	UF : 1, UT : 1,		CONFIG : 'N U T, 0, 0, 1',
	X =  112.000  mm,	Y =  46.000  mm,	Z =   0.600 mm,
	W =180.000 deg,	P =   0.000 deg,	R =    90.000 deg
};
P[2787]{
   GP1:
	UF : 1, UT : 1,		CONFIG : 'N U T, 0, 0, 1',
	X =  112.000  mm,	Y =  46.000  mm,	Z =   15.000 mm,
	W =180.000 deg,	P =   0.000 deg,	R =    90.000 deg
};
P[2794]{
   GP1:
	UF : 1, UT : 1,		CONFIG : 'N U T, 0, 0, 1',
	X =  127.000  mm,	Y =  46.000  mm,	Z =   15.000 mm,
	W =180.000 deg,	P =   0.000 deg,	R =    90.000 deg
};
P[2795]{
   GP1:
	UF : 1, UT : 1,		CONFIG : 'N U T, 0, 0, 1',
	X =  127.000  mm,	Y =  46.000  mm,	Z =   0.600 mm,
	W =180.000 deg,	P =   0.000 deg,	R =    90.000 deg
};
P[2796]{
   GP1:
	UF : 1, UT : 1,		CONFIG : 'N U T, 0, 0, 1',
	X =  127.000  mm,	Y =  46.000  mm,	Z =   15.000 mm,
	W =180.000 deg,	P =   0.000 deg,	R =    90.000 deg
};
P[2797]{
   GP1:
	UF : 1, UT : 1,		CONFIG : 'N U T, 0, 0, 1',
	X =  130.000  mm,	Y =  46.000  mm,	Z =   15.000 mm,
	W =180.000 deg,	P =   0.000 deg,	R =    90.000 deg
};
P[2798]{
   GP1:
	UF : 1, UT : 1,		CONFIG : 'N U T, 0, 0, 1',
	X =  130.000  mm,	Y =  46.000  mm,	Z =   0.600 mm,
	W =180.000 deg,	P =   0.000 deg,	R =    90.000 deg
};
P[2799]{
   GP1:
	UF : 1, UT : 1,		CONFIG : 'N U T, 0, 0, 1',
	X =  130.000  mm,	Y =  46.000  mm,	Z =   15.000 mm,
	W =180.000 deg,	P =   0.000 deg,	R =    90.000 deg
};
P[2800]{
   GP1:
	UF : 1, UT : 1,		CONFIG : 'N U T, 0, 0, 1',
	X =  133.000  mm,	Y =  46.000  mm,	Z =   15.000 mm,
	W =180.000 deg,	P =   0.000 deg,	R =    90.000 deg
};
P[2801]{
   GP1:
	UF : 1, UT : 1,		CONFIG : 'N U T, 0, 0, 1',
	X =  133.000  mm,	Y =  46.000  mm,	Z =   0.600 mm,
	W =180.000 deg,	P =   0.000 deg,	R =    90.000 deg
};
P[2802]{
   GP1:
	UF : 1, UT : 1,		CONFIG : 'N U T, 0, 0, 1',
	X =  133.000  mm,	Y =  46.000  mm,	Z =   15.000 mm,
	W =180.000 deg,	P =   0.000 deg,	R =    90.000 deg
};
P[2806]{
   GP1:
	UF : 1, UT : 1,		CONFIG : 'N U T, 0, 0, 1',
	X =  139.000  mm,	Y =  46.000  mm,	Z =   15.000 mm,
	W =180.000 deg,	P =   0.000 deg,	R =    90.000 deg
};
P[2807]{
   GP1:
	UF : 1, UT : 1,		CONFIG : 'N U T, 0, 0, 1',
	X =  139.000  mm,	Y =  46.000  mm,	Z =   0.600 mm,
	W =180.000 deg,	P =   0.000 deg,	R =    90.000 deg
};
P[2808]{
   GP1:
	UF : 1, UT : 1,		CONFIG : 'N U T, 0, 0, 1',
	X =  139.000  mm,	Y =  46.000  mm,	Z =   15.000 mm,
	W =180.000 deg,	P =   0.000 deg,	R =    90.000 deg
};
P[2812]{
   GP1:
	UF : 1, UT : 1,		CONFIG : 'N U T, 0, 0, 1',
	X =  145.000  mm,	Y =  46.000  mm,	Z =   15.000 mm,
	W =180.000 deg,	P =   0.000 deg,	R =    90.000 deg
};
P[2813]{
   GP1:
	UF : 1, UT : 1,		CONFIG : 'N U T, 0, 0, 1',
	X =  145.000  mm,	Y =  46.000  mm,	Z =   0.600 mm,
	W =180.000 deg,	P =   0.000 deg,	R =    90.000 deg
};
P[2814]{
   GP1:
	UF : 1, UT : 1,		CONFIG : 'N U T, 0, 0, 1',
	X =  145.000  mm,	Y =  46.000  mm,	Z =   15.000 mm,
	W =180.000 deg,	P =   0.000 deg,	R =    90.000 deg
};
P[2824]{
   GP1:
	UF : 1, UT : 1,		CONFIG : 'N U T, 0, 0, 1',
	X =  175.000  mm,	Y =  46.000  mm,	Z =   15.000 mm,
	W =180.000 deg,	P =   0.000 deg,	R =    90.000 deg
};
P[2825]{
   GP1:
	UF : 1, UT : 1,		CONFIG : 'N U T, 0, 0, 1',
	X =  175.000  mm,	Y =  46.000  mm,	Z =   0.600 mm,
	W =180.000 deg,	P =   0.000 deg,	R =    90.000 deg
};
P[2826]{
   GP1:
	UF : 1, UT : 1,		CONFIG : 'N U T, 0, 0, 1',
	X =  175.000  mm,	Y =  46.000  mm,	Z =   15.000 mm,
	W =180.000 deg,	P =   0.000 deg,	R =    90.000 deg
};
P[2827]{
   GP1:
	UF : 1, UT : 1,		CONFIG : 'N U T, 0, 0, 1',
	X =  178.000  mm,	Y =  46.000  mm,	Z =   15.000 mm,
	W =180.000 deg,	P =   0.000 deg,	R =    90.000 deg
};
P[2828]{
   GP1:
	UF : 1, UT : 1,		CONFIG : 'N U T, 0, 0, 1',
	X =  178.000  mm,	Y =  46.000  mm,	Z =   0.600 mm,
	W =180.000 deg,	P =   0.000 deg,	R =    90.000 deg
};
P[2829]{
   GP1:
	UF : 1, UT : 1,		CONFIG : 'N U T, 0, 0, 1',
	X =  178.000  mm,	Y =  46.000  mm,	Z =   15.000 mm,
	W =180.000 deg,	P =   0.000 deg,	R =    90.000 deg
};
P[2830]{
   GP1:
	UF : 1, UT : 1,		CONFIG : 'N U T, 0, 0, 1',
	X =  1.000  mm,	Y =  49.000  mm,	Z =   15.000 mm,
	W =180.000 deg,	P =   0.000 deg,	R =    90.000 deg
};
P[2831]{
   GP1:
	UF : 1, UT : 1,		CONFIG : 'N U T, 0, 0, 1',
	X =  1.000  mm,	Y =  49.000  mm,	Z =   0.600 mm,
	W =180.000 deg,	P =   0.000 deg,	R =    90.000 deg
};
P[2832]{
   GP1:
	UF : 1, UT : 1,		CONFIG : 'N U T, 0, 0, 1',
	X =  1.000  mm,	Y =  49.000  mm,	Z =   15.000 mm,
	W =180.000 deg,	P =   0.000 deg,	R =    90.000 deg
};
P[2833]{
   GP1:
	UF : 1, UT : 1,		CONFIG : 'N U T, 0, 0, 1',
	X =  4.000  mm,	Y =  49.000  mm,	Z =   15.000 mm,
	W =180.000 deg,	P =   0.000 deg,	R =    90.000 deg
};
P[2834]{
   GP1:
	UF : 1, UT : 1,		CONFIG : 'N U T, 0, 0, 1',
	X =  4.000  mm,	Y =  49.000  mm,	Z =   0.600 mm,
	W =180.000 deg,	P =   0.000 deg,	R =    90.000 deg
};
P[2835]{
   GP1:
	UF : 1, UT : 1,		CONFIG : 'N U T, 0, 0, 1',
	X =  4.000  mm,	Y =  49.000  mm,	Z =   15.000 mm,
	W =180.000 deg,	P =   0.000 deg,	R =    90.000 deg
};
P[2836]{
   GP1:
	UF : 1, UT : 1,		CONFIG : 'N U T, 0, 0, 1',
	X =  7.000  mm,	Y =  49.000  mm,	Z =   15.000 mm,
	W =180.000 deg,	P =   0.000 deg,	R =    90.000 deg
};
P[2837]{
   GP1:
	UF : 1, UT : 1,		CONFIG : 'N U T, 0, 0, 1',
	X =  7.000  mm,	Y =  49.000  mm,	Z =   0.600 mm,
	W =180.000 deg,	P =   0.000 deg,	R =    90.000 deg
};
P[2838]{
   GP1:
	UF : 1, UT : 1,		CONFIG : 'N U T, 0, 0, 1',
	X =  7.000  mm,	Y =  49.000  mm,	Z =   15.000 mm,
	W =180.000 deg,	P =   0.000 deg,	R =    90.000 deg
};
P[2839]{
   GP1:
	UF : 1, UT : 1,		CONFIG : 'N U T, 0, 0, 1',
	X =  10.000  mm,	Y =  49.000  mm,	Z =   15.000 mm,
	W =180.000 deg,	P =   0.000 deg,	R =    90.000 deg
};
P[2840]{
   GP1:
	UF : 1, UT : 1,		CONFIG : 'N U T, 0, 0, 1',
	X =  10.000  mm,	Y =  49.000  mm,	Z =   0.600 mm,
	W =180.000 deg,	P =   0.000 deg,	R =    90.000 deg
};
P[2841]{
   GP1:
	UF : 1, UT : 1,		CONFIG : 'N U T, 0, 0, 1',
	X =  10.000  mm,	Y =  49.000  mm,	Z =   15.000 mm,
	W =180.000 deg,	P =   0.000 deg,	R =    90.000 deg
};
P[2842]{
   GP1:
	UF : 1, UT : 1,		CONFIG : 'N U T, 0, 0, 1',
	X =  13.000  mm,	Y =  49.000  mm,	Z =   15.000 mm,
	W =180.000 deg,	P =   0.000 deg,	R =    90.000 deg
};
P[2843]{
   GP1:
	UF : 1, UT : 1,		CONFIG : 'N U T, 0, 0, 1',
	X =  13.000  mm,	Y =  49.000  mm,	Z =   0.600 mm,
	W =180.000 deg,	P =   0.000 deg,	R =    90.000 deg
};
P[2844]{
   GP1:
	UF : 1, UT : 1,		CONFIG : 'N U T, 0, 0, 1',
	X =  13.000  mm,	Y =  49.000  mm,	Z =   15.000 mm,
	W =180.000 deg,	P =   0.000 deg,	R =    90.000 deg
};
P[2845]{
   GP1:
	UF : 1, UT : 1,		CONFIG : 'N U T, 0, 0, 1',
	X =  16.000  mm,	Y =  49.000  mm,	Z =   15.000 mm,
	W =180.000 deg,	P =   0.000 deg,	R =    90.000 deg
};
P[2846]{
   GP1:
	UF : 1, UT : 1,		CONFIG : 'N U T, 0, 0, 1',
	X =  16.000  mm,	Y =  49.000  mm,	Z =   0.600 mm,
	W =180.000 deg,	P =   0.000 deg,	R =    90.000 deg
};
P[2847]{
   GP1:
	UF : 1, UT : 1,		CONFIG : 'N U T, 0, 0, 1',
	X =  16.000  mm,	Y =  49.000  mm,	Z =   15.000 mm,
	W =180.000 deg,	P =   0.000 deg,	R =    90.000 deg
};
P[2848]{
   GP1:
	UF : 1, UT : 1,		CONFIG : 'N U T, 0, 0, 1',
	X =  19.000  mm,	Y =  49.000  mm,	Z =   15.000 mm,
	W =180.000 deg,	P =   0.000 deg,	R =    90.000 deg
};
P[2849]{
   GP1:
	UF : 1, UT : 1,		CONFIG : 'N U T, 0, 0, 1',
	X =  19.000  mm,	Y =  49.000  mm,	Z =   0.600 mm,
	W =180.000 deg,	P =   0.000 deg,	R =    90.000 deg
};
P[2850]{
   GP1:
	UF : 1, UT : 1,		CONFIG : 'N U T, 0, 0, 1',
	X =  19.000  mm,	Y =  49.000  mm,	Z =   15.000 mm,
	W =180.000 deg,	P =   0.000 deg,	R =    90.000 deg
};
P[2854]{
   GP1:
	UF : 1, UT : 1,		CONFIG : 'N U T, 0, 0, 1',
	X =  25.000  mm,	Y =  49.000  mm,	Z =   15.000 mm,
	W =180.000 deg,	P =   0.000 deg,	R =    90.000 deg
};
P[2855]{
   GP1:
	UF : 1, UT : 1,		CONFIG : 'N U T, 0, 0, 1',
	X =  25.000  mm,	Y =  49.000  mm,	Z =   0.600 mm,
	W =180.000 deg,	P =   0.000 deg,	R =    90.000 deg
};
P[2856]{
   GP1:
	UF : 1, UT : 1,		CONFIG : 'N U T, 0, 0, 1',
	X =  25.000  mm,	Y =  49.000  mm,	Z =   15.000 mm,
	W =180.000 deg,	P =   0.000 deg,	R =    90.000 deg
};
P[2857]{
   GP1:
	UF : 1, UT : 1,		CONFIG : 'N U T, 0, 0, 1',
	X =  28.000  mm,	Y =  49.000  mm,	Z =   15.000 mm,
	W =180.000 deg,	P =   0.000 deg,	R =    90.000 deg
};
P[2858]{
   GP1:
	UF : 1, UT : 1,		CONFIG : 'N U T, 0, 0, 1',
	X =  28.000  mm,	Y =  49.000  mm,	Z =   0.600 mm,
	W =180.000 deg,	P =   0.000 deg,	R =    90.000 deg
};
P[2859]{
   GP1:
	UF : 1, UT : 1,		CONFIG : 'N U T, 0, 0, 1',
	X =  28.000  mm,	Y =  49.000  mm,	Z =   15.000 mm,
	W =180.000 deg,	P =   0.000 deg,	R =    90.000 deg
};
P[2860]{
   GP1:
	UF : 1, UT : 1,		CONFIG : 'N U T, 0, 0, 1',
	X =  31.000  mm,	Y =  49.000  mm,	Z =   15.000 mm,
	W =180.000 deg,	P =   0.000 deg,	R =    90.000 deg
};
P[2861]{
   GP1:
	UF : 1, UT : 1,		CONFIG : 'N U T, 0, 0, 1',
	X =  31.000  mm,	Y =  49.000  mm,	Z =   0.600 mm,
	W =180.000 deg,	P =   0.000 deg,	R =    90.000 deg
};
P[2862]{
   GP1:
	UF : 1, UT : 1,		CONFIG : 'N U T, 0, 0, 1',
	X =  31.000  mm,	Y =  49.000  mm,	Z =   15.000 mm,
	W =180.000 deg,	P =   0.000 deg,	R =    90.000 deg
};
P[2863]{
   GP1:
	UF : 1, UT : 1,		CONFIG : 'N U T, 0, 0, 1',
	X =  34.000  mm,	Y =  49.000  mm,	Z =   15.000 mm,
	W =180.000 deg,	P =   0.000 deg,	R =    90.000 deg
};
P[2864]{
   GP1:
	UF : 1, UT : 1,		CONFIG : 'N U T, 0, 0, 1',
	X =  34.000  mm,	Y =  49.000  mm,	Z =   0.600 mm,
	W =180.000 deg,	P =   0.000 deg,	R =    90.000 deg
};
P[2865]{
   GP1:
	UF : 1, UT : 1,		CONFIG : 'N U T, 0, 0, 1',
	X =  34.000  mm,	Y =  49.000  mm,	Z =   15.000 mm,
	W =180.000 deg,	P =   0.000 deg,	R =    90.000 deg
};
P[2866]{
   GP1:
	UF : 1, UT : 1,		CONFIG : 'N U T, 0, 0, 1',
	X =  37.000  mm,	Y =  49.000  mm,	Z =   15.000 mm,
	W =180.000 deg,	P =   0.000 deg,	R =    90.000 deg
};
P[2867]{
   GP1:
	UF : 1, UT : 1,		CONFIG : 'N U T, 0, 0, 1',
	X =  37.000  mm,	Y =  49.000  mm,	Z =   0.600 mm,
	W =180.000 deg,	P =   0.000 deg,	R =    90.000 deg
};
P[2868]{
   GP1:
	UF : 1, UT : 1,		CONFIG : 'N U T, 0, 0, 1',
	X =  37.000  mm,	Y =  49.000  mm,	Z =   15.000 mm,
	W =180.000 deg,	P =   0.000 deg,	R =    90.000 deg
};
P[2869]{
   GP1:
	UF : 1, UT : 1,		CONFIG : 'N U T, 0, 0, 1',
	X =  40.000  mm,	Y =  49.000  mm,	Z =   15.000 mm,
	W =180.000 deg,	P =   0.000 deg,	R =    90.000 deg
};
P[2870]{
   GP1:
	UF : 1, UT : 1,		CONFIG : 'N U T, 0, 0, 1',
	X =  40.000  mm,	Y =  49.000  mm,	Z =   0.600 mm,
	W =180.000 deg,	P =   0.000 deg,	R =    90.000 deg
};
P[2871]{
   GP1:
	UF : 1, UT : 1,		CONFIG : 'N U T, 0, 0, 1',
	X =  40.000  mm,	Y =  49.000  mm,	Z =   15.000 mm,
	W =180.000 deg,	P =   0.000 deg,	R =    90.000 deg
};
P[2872]{
   GP1:
	UF : 1, UT : 1,		CONFIG : 'N U T, 0, 0, 1',
	X =  43.000  mm,	Y =  49.000  mm,	Z =   15.000 mm,
	W =180.000 deg,	P =   0.000 deg,	R =    90.000 deg
};
P[2873]{
   GP1:
	UF : 1, UT : 1,		CONFIG : 'N U T, 0, 0, 1',
	X =  43.000  mm,	Y =  49.000  mm,	Z =   0.600 mm,
	W =180.000 deg,	P =   0.000 deg,	R =    90.000 deg
};
P[2874]{
   GP1:
	UF : 1, UT : 1,		CONFIG : 'N U T, 0, 0, 1',
	X =  43.000  mm,	Y =  49.000  mm,	Z =   15.000 mm,
	W =180.000 deg,	P =   0.000 deg,	R =    90.000 deg
};
P[2875]{
   GP1:
	UF : 1, UT : 1,		CONFIG : 'N U T, 0, 0, 1',
	X =  46.000  mm,	Y =  49.000  mm,	Z =   15.000 mm,
	W =180.000 deg,	P =   0.000 deg,	R =    90.000 deg
};
P[2876]{
   GP1:
	UF : 1, UT : 1,		CONFIG : 'N U T, 0, 0, 1',
	X =  46.000  mm,	Y =  49.000  mm,	Z =   0.600 mm,
	W =180.000 deg,	P =   0.000 deg,	R =    90.000 deg
};
P[2877]{
   GP1:
	UF : 1, UT : 1,		CONFIG : 'N U T, 0, 0, 1',
	X =  46.000  mm,	Y =  49.000  mm,	Z =   15.000 mm,
	W =180.000 deg,	P =   0.000 deg,	R =    90.000 deg
};
P[2878]{
   GP1:
	UF : 1, UT : 1,		CONFIG : 'N U T, 0, 0, 1',
	X =  49.000  mm,	Y =  49.000  mm,	Z =   15.000 mm,
	W =180.000 deg,	P =   0.000 deg,	R =    90.000 deg
};
P[2879]{
   GP1:
	UF : 1, UT : 1,		CONFIG : 'N U T, 0, 0, 1',
	X =  49.000  mm,	Y =  49.000  mm,	Z =   0.600 mm,
	W =180.000 deg,	P =   0.000 deg,	R =    90.000 deg
};
P[2880]{
   GP1:
	UF : 1, UT : 1,		CONFIG : 'N U T, 0, 0, 1',
	X =  49.000  mm,	Y =  49.000  mm,	Z =   15.000 mm,
	W =180.000 deg,	P =   0.000 deg,	R =    90.000 deg
};
P[2881]{
   GP1:
	UF : 1, UT : 1,		CONFIG : 'N U T, 0, 0, 1',
	X =  52.000  mm,	Y =  49.000  mm,	Z =   15.000 mm,
	W =180.000 deg,	P =   0.000 deg,	R =    90.000 deg
};
P[2882]{
   GP1:
	UF : 1, UT : 1,		CONFIG : 'N U T, 0, 0, 1',
	X =  52.000  mm,	Y =  49.000  mm,	Z =   0.600 mm,
	W =180.000 deg,	P =   0.000 deg,	R =    90.000 deg
};
P[2883]{
   GP1:
	UF : 1, UT : 1,		CONFIG : 'N U T, 0, 0, 1',
	X =  52.000  mm,	Y =  49.000  mm,	Z =   15.000 mm,
	W =180.000 deg,	P =   0.000 deg,	R =    90.000 deg
};
P[2884]{
   GP1:
	UF : 1, UT : 1,		CONFIG : 'N U T, 0, 0, 1',
	X =  55.000  mm,	Y =  49.000  mm,	Z =   15.000 mm,
	W =180.000 deg,	P =   0.000 deg,	R =    90.000 deg
};
P[2885]{
   GP1:
	UF : 1, UT : 1,		CONFIG : 'N U T, 0, 0, 1',
	X =  55.000  mm,	Y =  49.000  mm,	Z =   0.600 mm,
	W =180.000 deg,	P =   0.000 deg,	R =    90.000 deg
};
P[2886]{
   GP1:
	UF : 1, UT : 1,		CONFIG : 'N U T, 0, 0, 1',
	X =  55.000  mm,	Y =  49.000  mm,	Z =   15.000 mm,
	W =180.000 deg,	P =   0.000 deg,	R =    90.000 deg
};
P[2887]{
   GP1:
	UF : 1, UT : 1,		CONFIG : 'N U T, 0, 0, 1',
	X =  58.000  mm,	Y =  49.000  mm,	Z =   15.000 mm,
	W =180.000 deg,	P =   0.000 deg,	R =    90.000 deg
};
P[2888]{
   GP1:
	UF : 1, UT : 1,		CONFIG : 'N U T, 0, 0, 1',
	X =  58.000  mm,	Y =  49.000  mm,	Z =   0.600 mm,
	W =180.000 deg,	P =   0.000 deg,	R =    90.000 deg
};
P[2889]{
   GP1:
	UF : 1, UT : 1,		CONFIG : 'N U T, 0, 0, 1',
	X =  58.000  mm,	Y =  49.000  mm,	Z =   15.000 mm,
	W =180.000 deg,	P =   0.000 deg,	R =    90.000 deg
};
P[2899]{
   GP1:
	UF : 1, UT : 1,		CONFIG : 'N U T, 0, 0, 1',
	X =  70.000  mm,	Y =  49.000  mm,	Z =   15.000 mm,
	W =180.000 deg,	P =   0.000 deg,	R =    90.000 deg
};
P[2900]{
   GP1:
	UF : 1, UT : 1,		CONFIG : 'N U T, 0, 0, 1',
	X =  70.000  mm,	Y =  49.000  mm,	Z =   0.600 mm,
	W =180.000 deg,	P =   0.000 deg,	R =    90.000 deg
};
P[2901]{
   GP1:
	UF : 1, UT : 1,		CONFIG : 'N U T, 0, 0, 1',
	X =  70.000  mm,	Y =  49.000  mm,	Z =   15.000 mm,
	W =180.000 deg,	P =   0.000 deg,	R =    90.000 deg
};
P[2902]{
   GP1:
	UF : 1, UT : 1,		CONFIG : 'N U T, 0, 0, 1',
	X =  73.000  mm,	Y =  49.000  mm,	Z =   15.000 mm,
	W =180.000 deg,	P =   0.000 deg,	R =    90.000 deg
};
P[2903]{
   GP1:
	UF : 1, UT : 1,		CONFIG : 'N U T, 0, 0, 1',
	X =  73.000  mm,	Y =  49.000  mm,	Z =   0.600 mm,
	W =180.000 deg,	P =   0.000 deg,	R =    90.000 deg
};
P[2904]{
   GP1:
	UF : 1, UT : 1,		CONFIG : 'N U T, 0, 0, 1',
	X =  73.000  mm,	Y =  49.000  mm,	Z =   15.000 mm,
	W =180.000 deg,	P =   0.000 deg,	R =    90.000 deg
};
P[2905]{
   GP1:
	UF : 1, UT : 1,		CONFIG : 'N U T, 0, 0, 1',
	X =  76.000  mm,	Y =  49.000  mm,	Z =   15.000 mm,
	W =180.000 deg,	P =   0.000 deg,	R =    90.000 deg
};
P[2906]{
   GP1:
	UF : 1, UT : 1,		CONFIG : 'N U T, 0, 0, 1',
	X =  76.000  mm,	Y =  49.000  mm,	Z =   0.600 mm,
	W =180.000 deg,	P =   0.000 deg,	R =    90.000 deg
};
P[2907]{
   GP1:
	UF : 1, UT : 1,		CONFIG : 'N U T, 0, 0, 1',
	X =  76.000  mm,	Y =  49.000  mm,	Z =   15.000 mm,
	W =180.000 deg,	P =   0.000 deg,	R =    90.000 deg
};
P[2917]{
   GP1:
	UF : 1, UT : 1,		CONFIG : 'N U T, 0, 0, 1',
	X =  88.000  mm,	Y =  49.000  mm,	Z =   15.000 mm,
	W =180.000 deg,	P =   0.000 deg,	R =    90.000 deg
};
P[2918]{
   GP1:
	UF : 1, UT : 1,		CONFIG : 'N U T, 0, 0, 1',
	X =  88.000  mm,	Y =  49.000  mm,	Z =   0.600 mm,
	W =180.000 deg,	P =   0.000 deg,	R =    90.000 deg
};
P[2919]{
   GP1:
	UF : 1, UT : 1,		CONFIG : 'N U T, 0, 0, 1',
	X =  88.000  mm,	Y =  49.000  mm,	Z =   15.000 mm,
	W =180.000 deg,	P =   0.000 deg,	R =    90.000 deg
};
P[2920]{
   GP1:
	UF : 1, UT : 1,		CONFIG : 'N U T, 0, 0, 1',
	X =  91.000  mm,	Y =  49.000  mm,	Z =   15.000 mm,
	W =180.000 deg,	P =   0.000 deg,	R =    90.000 deg
};
P[2921]{
   GP1:
	UF : 1, UT : 1,		CONFIG : 'N U T, 0, 0, 1',
	X =  91.000  mm,	Y =  49.000  mm,	Z =   0.600 mm,
	W =180.000 deg,	P =   0.000 deg,	R =    90.000 deg
};
P[2922]{
   GP1:
	UF : 1, UT : 1,		CONFIG : 'N U T, 0, 0, 1',
	X =  91.000  mm,	Y =  49.000  mm,	Z =   15.000 mm,
	W =180.000 deg,	P =   0.000 deg,	R =    90.000 deg
};
P[2923]{
   GP1:
	UF : 1, UT : 1,		CONFIG : 'N U T, 0, 0, 1',
	X =  94.000  mm,	Y =  49.000  mm,	Z =   15.000 mm,
	W =180.000 deg,	P =   0.000 deg,	R =    90.000 deg
};
P[2924]{
   GP1:
	UF : 1, UT : 1,		CONFIG : 'N U T, 0, 0, 1',
	X =  94.000  mm,	Y =  49.000  mm,	Z =   0.600 mm,
	W =180.000 deg,	P =   0.000 deg,	R =    90.000 deg
};
P[2925]{
   GP1:
	UF : 1, UT : 1,		CONFIG : 'N U T, 0, 0, 1',
	X =  94.000  mm,	Y =  49.000  mm,	Z =   15.000 mm,
	W =180.000 deg,	P =   0.000 deg,	R =    90.000 deg
};
P[2926]{
   GP1:
	UF : 1, UT : 1,		CONFIG : 'N U T, 0, 0, 1',
	X =  97.000  mm,	Y =  49.000  mm,	Z =   15.000 mm,
	W =180.000 deg,	P =   0.000 deg,	R =    90.000 deg
};
P[2927]{
   GP1:
	UF : 1, UT : 1,		CONFIG : 'N U T, 0, 0, 1',
	X =  97.000  mm,	Y =  49.000  mm,	Z =   0.600 mm,
	W =180.000 deg,	P =   0.000 deg,	R =    90.000 deg
};
P[2928]{
   GP1:
	UF : 1, UT : 1,		CONFIG : 'N U T, 0, 0, 1',
	X =  97.000  mm,	Y =  49.000  mm,	Z =   15.000 mm,
	W =180.000 deg,	P =   0.000 deg,	R =    90.000 deg
};
P[2929]{
   GP1:
	UF : 1, UT : 1,		CONFIG : 'N U T, 0, 0, 1',
	X =  100.000  mm,	Y =  49.000  mm,	Z =   15.000 mm,
	W =180.000 deg,	P =   0.000 deg,	R =    90.000 deg
};
P[2930]{
   GP1:
	UF : 1, UT : 1,		CONFIG : 'N U T, 0, 0, 1',
	X =  100.000  mm,	Y =  49.000  mm,	Z =   0.600 mm,
	W =180.000 deg,	P =   0.000 deg,	R =    90.000 deg
};
P[2931]{
   GP1:
	UF : 1, UT : 1,		CONFIG : 'N U T, 0, 0, 1',
	X =  100.000  mm,	Y =  49.000  mm,	Z =   15.000 mm,
	W =180.000 deg,	P =   0.000 deg,	R =    90.000 deg
};
P[2932]{
   GP1:
	UF : 1, UT : 1,		CONFIG : 'N U T, 0, 0, 1',
	X =  103.000  mm,	Y =  49.000  mm,	Z =   15.000 mm,
	W =180.000 deg,	P =   0.000 deg,	R =    90.000 deg
};
P[2933]{
   GP1:
	UF : 1, UT : 1,		CONFIG : 'N U T, 0, 0, 1',
	X =  103.000  mm,	Y =  49.000  mm,	Z =   0.600 mm,
	W =180.000 deg,	P =   0.000 deg,	R =    90.000 deg
};
P[2934]{
   GP1:
	UF : 1, UT : 1,		CONFIG : 'N U T, 0, 0, 1',
	X =  103.000  mm,	Y =  49.000  mm,	Z =   15.000 mm,
	W =180.000 deg,	P =   0.000 deg,	R =    90.000 deg
};
P[2935]{
   GP1:
	UF : 1, UT : 1,		CONFIG : 'N U T, 0, 0, 1',
	X =  106.000  mm,	Y =  49.000  mm,	Z =   15.000 mm,
	W =180.000 deg,	P =   0.000 deg,	R =    90.000 deg
};
P[2936]{
   GP1:
	UF : 1, UT : 1,		CONFIG : 'N U T, 0, 0, 1',
	X =  106.000  mm,	Y =  49.000  mm,	Z =   0.600 mm,
	W =180.000 deg,	P =   0.000 deg,	R =    90.000 deg
};
P[2937]{
   GP1:
	UF : 1, UT : 1,		CONFIG : 'N U T, 0, 0, 1',
	X =  106.000  mm,	Y =  49.000  mm,	Z =   15.000 mm,
	W =180.000 deg,	P =   0.000 deg,	R =    90.000 deg
};
P[2938]{
   GP1:
	UF : 1, UT : 1,		CONFIG : 'N U T, 0, 0, 1',
	X =  109.000  mm,	Y =  49.000  mm,	Z =   15.000 mm,
	W =180.000 deg,	P =   0.000 deg,	R =    90.000 deg
};
P[2939]{
   GP1:
	UF : 1, UT : 1,		CONFIG : 'N U T, 0, 0, 1',
	X =  109.000  mm,	Y =  49.000  mm,	Z =   0.600 mm,
	W =180.000 deg,	P =   0.000 deg,	R =    90.000 deg
};
P[2940]{
   GP1:
	UF : 1, UT : 1,		CONFIG : 'N U T, 0, 0, 1',
	X =  109.000  mm,	Y =  49.000  mm,	Z =   15.000 mm,
	W =180.000 deg,	P =   0.000 deg,	R =    90.000 deg
};
P[2941]{
   GP1:
	UF : 1, UT : 1,		CONFIG : 'N U T, 0, 0, 1',
	X =  112.000  mm,	Y =  49.000  mm,	Z =   15.000 mm,
	W =180.000 deg,	P =   0.000 deg,	R =    90.000 deg
};
P[2942]{
   GP1:
	UF : 1, UT : 1,		CONFIG : 'N U T, 0, 0, 1',
	X =  112.000  mm,	Y =  49.000  mm,	Z =   0.600 mm,
	W =180.000 deg,	P =   0.000 deg,	R =    90.000 deg
};
P[2943]{
   GP1:
	UF : 1, UT : 1,		CONFIG : 'N U T, 0, 0, 1',
	X =  112.000  mm,	Y =  49.000  mm,	Z =   15.000 mm,
	W =180.000 deg,	P =   0.000 deg,	R =    90.000 deg
};
P[2950]{
   GP1:
	UF : 1, UT : 1,		CONFIG : 'N U T, 0, 0, 1',
	X =  127.000  mm,	Y =  49.000  mm,	Z =   15.000 mm,
	W =180.000 deg,	P =   0.000 deg,	R =    90.000 deg
};
P[2951]{
   GP1:
	UF : 1, UT : 1,		CONFIG : 'N U T, 0, 0, 1',
	X =  127.000  mm,	Y =  49.000  mm,	Z =   0.600 mm,
	W =180.000 deg,	P =   0.000 deg,	R =    90.000 deg
};
P[2952]{
   GP1:
	UF : 1, UT : 1,		CONFIG : 'N U T, 0, 0, 1',
	X =  127.000  mm,	Y =  49.000  mm,	Z =   15.000 mm,
	W =180.000 deg,	P =   0.000 deg,	R =    90.000 deg
};
P[2953]{
   GP1:
	UF : 1, UT : 1,		CONFIG : 'N U T, 0, 0, 1',
	X =  130.000  mm,	Y =  49.000  mm,	Z =   15.000 mm,
	W =180.000 deg,	P =   0.000 deg,	R =    90.000 deg
};
P[2954]{
   GP1:
	UF : 1, UT : 1,		CONFIG : 'N U T, 0, 0, 1',
	X =  130.000  mm,	Y =  49.000  mm,	Z =   0.600 mm,
	W =180.000 deg,	P =   0.000 deg,	R =    90.000 deg
};
P[2955]{
   GP1:
	UF : 1, UT : 1,		CONFIG : 'N U T, 0, 0, 1',
	X =  130.000  mm,	Y =  49.000  mm,	Z =   15.000 mm,
	W =180.000 deg,	P =   0.000 deg,	R =    90.000 deg
};
P[2959]{
   GP1:
	UF : 1, UT : 1,		CONFIG : 'N U T, 0, 0, 1',
	X =  136.000  mm,	Y =  49.000  mm,	Z =   15.000 mm,
	W =180.000 deg,	P =   0.000 deg,	R =    90.000 deg
};
P[2960]{
   GP1:
	UF : 1, UT : 1,		CONFIG : 'N U T, 0, 0, 1',
	X =  136.000  mm,	Y =  49.000  mm,	Z =   0.600 mm,
	W =180.000 deg,	P =   0.000 deg,	R =    90.000 deg
};
P[2961]{
   GP1:
	UF : 1, UT : 1,		CONFIG : 'N U T, 0, 0, 1',
	X =  136.000  mm,	Y =  49.000  mm,	Z =   15.000 mm,
	W =180.000 deg,	P =   0.000 deg,	R =    90.000 deg
};
P[2965]{
   GP1:
	UF : 1, UT : 1,		CONFIG : 'N U T, 0, 0, 1',
	X =  142.000  mm,	Y =  49.000  mm,	Z =   15.000 mm,
	W =180.000 deg,	P =   0.000 deg,	R =    90.000 deg
};
P[2966]{
   GP1:
	UF : 1, UT : 1,		CONFIG : 'N U T, 0, 0, 1',
	X =  142.000  mm,	Y =  49.000  mm,	Z =   0.600 mm,
	W =180.000 deg,	P =   0.000 deg,	R =    90.000 deg
};
P[2967]{
   GP1:
	UF : 1, UT : 1,		CONFIG : 'N U T, 0, 0, 1',
	X =  142.000  mm,	Y =  49.000  mm,	Z =   15.000 mm,
	W =180.000 deg,	P =   0.000 deg,	R =    90.000 deg
};
P[2986]{
   GP1:
	UF : 1, UT : 1,		CONFIG : 'N U T, 0, 0, 1',
	X =  175.000  mm,	Y =  49.000  mm,	Z =   15.000 mm,
	W =180.000 deg,	P =   0.000 deg,	R =    90.000 deg
};
P[2987]{
   GP1:
	UF : 1, UT : 1,		CONFIG : 'N U T, 0, 0, 1',
	X =  175.000  mm,	Y =  49.000  mm,	Z =   0.600 mm,
	W =180.000 deg,	P =   0.000 deg,	R =    90.000 deg
};
P[2988]{
   GP1:
	UF : 1, UT : 1,		CONFIG : 'N U T, 0, 0, 1',
	X =  175.000  mm,	Y =  49.000  mm,	Z =   15.000 mm,
	W =180.000 deg,	P =   0.000 deg,	R =    90.000 deg
};
P[2989]{
   GP1:
	UF : 1, UT : 1,		CONFIG : 'N U T, 0, 0, 1',
	X =  178.000  mm,	Y =  49.000  mm,	Z =   15.000 mm,
	W =180.000 deg,	P =   0.000 deg,	R =    90.000 deg
};
P[2990]{
   GP1:
	UF : 1, UT : 1,		CONFIG : 'N U T, 0, 0, 1',
	X =  178.000  mm,	Y =  49.000  mm,	Z =   0.600 mm,
	W =180.000 deg,	P =   0.000 deg,	R =    90.000 deg
};
P[2991]{
   GP1:
	UF : 1, UT : 1,		CONFIG : 'N U T, 0, 0, 1',
	X =  178.000  mm,	Y =  49.000  mm,	Z =   15.000 mm,
	W =180.000 deg,	P =   0.000 deg,	R =    90.000 deg
};
P[2992]{
   GP1:
	UF : 1, UT : 1,		CONFIG : 'N U T, 0, 0, 1',
	X =  1.000  mm,	Y =  52.000  mm,	Z =   15.000 mm,
	W =180.000 deg,	P =   0.000 deg,	R =    90.000 deg
};
P[2993]{
   GP1:
	UF : 1, UT : 1,		CONFIG : 'N U T, 0, 0, 1',
	X =  1.000  mm,	Y =  52.000  mm,	Z =   0.600 mm,
	W =180.000 deg,	P =   0.000 deg,	R =    90.000 deg
};
P[2994]{
   GP1:
	UF : 1, UT : 1,		CONFIG : 'N U T, 0, 0, 1',
	X =  1.000  mm,	Y =  52.000  mm,	Z =   15.000 mm,
	W =180.000 deg,	P =   0.000 deg,	R =    90.000 deg
};
P[2995]{
   GP1:
	UF : 1, UT : 1,		CONFIG : 'N U T, 0, 0, 1',
	X =  4.000  mm,	Y =  52.000  mm,	Z =   15.000 mm,
	W =180.000 deg,	P =   0.000 deg,	R =    90.000 deg
};
P[2996]{
   GP1:
	UF : 1, UT : 1,		CONFIG : 'N U T, 0, 0, 1',
	X =  4.000  mm,	Y =  52.000  mm,	Z =   0.600 mm,
	W =180.000 deg,	P =   0.000 deg,	R =    90.000 deg
};
P[2997]{
   GP1:
	UF : 1, UT : 1,		CONFIG : 'N U T, 0, 0, 1',
	X =  4.000  mm,	Y =  52.000  mm,	Z =   15.000 mm,
	W =180.000 deg,	P =   0.000 deg,	R =    90.000 deg
};
P[2998]{
   GP1:
	UF : 1, UT : 1,		CONFIG : 'N U T, 0, 0, 1',
	X =  7.000  mm,	Y =  52.000  mm,	Z =   15.000 mm,
	W =180.000 deg,	P =   0.000 deg,	R =    90.000 deg
};
P[2999]{
   GP1:
	UF : 1, UT : 1,		CONFIG : 'N U T, 0, 0, 1',
	X =  7.000  mm,	Y =  52.000  mm,	Z =   0.600 mm,
	W =180.000 deg,	P =   0.000 deg,	R =    90.000 deg
};
P[3000]{
   GP1:
	UF : 1, UT : 1,		CONFIG : 'N U T, 0, 0, 1',
	X =  7.000  mm,	Y =  52.000  mm,	Z =   15.000 mm,
	W =180.000 deg,	P =   0.000 deg,	R =    90.000 deg
};
P[3001]{
   GP1:
	UF : 1, UT : 1,		CONFIG : 'N U T, 0, 0, 1',
	X =  10.000  mm,	Y =  52.000  mm,	Z =   15.000 mm,
	W =180.000 deg,	P =   0.000 deg,	R =    90.000 deg
};
P[3002]{
   GP1:
	UF : 1, UT : 1,		CONFIG : 'N U T, 0, 0, 1',
	X =  10.000  mm,	Y =  52.000  mm,	Z =   0.600 mm,
	W =180.000 deg,	P =   0.000 deg,	R =    90.000 deg
};
P[3003]{
   GP1:
	UF : 1, UT : 1,		CONFIG : 'N U T, 0, 0, 1',
	X =  10.000  mm,	Y =  52.000  mm,	Z =   15.000 mm,
	W =180.000 deg,	P =   0.000 deg,	R =    90.000 deg
};
P[3004]{
   GP1:
	UF : 1, UT : 1,		CONFIG : 'N U T, 0, 0, 1',
	X =  13.000  mm,	Y =  52.000  mm,	Z =   15.000 mm,
	W =180.000 deg,	P =   0.000 deg,	R =    90.000 deg
};
P[3005]{
   GP1:
	UF : 1, UT : 1,		CONFIG : 'N U T, 0, 0, 1',
	X =  13.000  mm,	Y =  52.000  mm,	Z =   0.600 mm,
	W =180.000 deg,	P =   0.000 deg,	R =    90.000 deg
};
P[3006]{
   GP1:
	UF : 1, UT : 1,		CONFIG : 'N U T, 0, 0, 1',
	X =  13.000  mm,	Y =  52.000  mm,	Z =   15.000 mm,
	W =180.000 deg,	P =   0.000 deg,	R =    90.000 deg
};
P[3007]{
   GP1:
	UF : 1, UT : 1,		CONFIG : 'N U T, 0, 0, 1',
	X =  16.000  mm,	Y =  52.000  mm,	Z =   15.000 mm,
	W =180.000 deg,	P =   0.000 deg,	R =    90.000 deg
};
P[3008]{
   GP1:
	UF : 1, UT : 1,		CONFIG : 'N U T, 0, 0, 1',
	X =  16.000  mm,	Y =  52.000  mm,	Z =   0.600 mm,
	W =180.000 deg,	P =   0.000 deg,	R =    90.000 deg
};
P[3009]{
   GP1:
	UF : 1, UT : 1,		CONFIG : 'N U T, 0, 0, 1',
	X =  16.000  mm,	Y =  52.000  mm,	Z =   15.000 mm,
	W =180.000 deg,	P =   0.000 deg,	R =    90.000 deg
};
P[3010]{
   GP1:
	UF : 1, UT : 1,		CONFIG : 'N U T, 0, 0, 1',
	X =  19.000  mm,	Y =  52.000  mm,	Z =   15.000 mm,
	W =180.000 deg,	P =   0.000 deg,	R =    90.000 deg
};
P[3011]{
   GP1:
	UF : 1, UT : 1,		CONFIG : 'N U T, 0, 0, 1',
	X =  19.000  mm,	Y =  52.000  mm,	Z =   0.600 mm,
	W =180.000 deg,	P =   0.000 deg,	R =    90.000 deg
};
P[3012]{
   GP1:
	UF : 1, UT : 1,		CONFIG : 'N U T, 0, 0, 1',
	X =  19.000  mm,	Y =  52.000  mm,	Z =   15.000 mm,
	W =180.000 deg,	P =   0.000 deg,	R =    90.000 deg
};
P[3013]{
   GP1:
	UF : 1, UT : 1,		CONFIG : 'N U T, 0, 0, 1',
	X =  25.000  mm,	Y =  52.000  mm,	Z =   15.000 mm,
	W =180.000 deg,	P =   0.000 deg,	R =    90.000 deg
};
P[3014]{
   GP1:
	UF : 1, UT : 1,		CONFIG : 'N U T, 0, 0, 1',
	X =  25.000  mm,	Y =  52.000  mm,	Z =   0.600 mm,
	W =180.000 deg,	P =   0.000 deg,	R =    90.000 deg
};
P[3015]{
   GP1:
	UF : 1, UT : 1,		CONFIG : 'N U T, 0, 0, 1',
	X =  25.000  mm,	Y =  52.000  mm,	Z =   15.000 mm,
	W =180.000 deg,	P =   0.000 deg,	R =    90.000 deg
};
P[3016]{
   GP1:
	UF : 1, UT : 1,		CONFIG : 'N U T, 0, 0, 1',
	X =  28.000  mm,	Y =  52.000  mm,	Z =   15.000 mm,
	W =180.000 deg,	P =   0.000 deg,	R =    90.000 deg
};
P[3017]{
   GP1:
	UF : 1, UT : 1,		CONFIG : 'N U T, 0, 0, 1',
	X =  28.000  mm,	Y =  52.000  mm,	Z =   0.600 mm,
	W =180.000 deg,	P =   0.000 deg,	R =    90.000 deg
};
P[3018]{
   GP1:
	UF : 1, UT : 1,		CONFIG : 'N U T, 0, 0, 1',
	X =  28.000  mm,	Y =  52.000  mm,	Z =   15.000 mm,
	W =180.000 deg,	P =   0.000 deg,	R =    90.000 deg
};
P[3019]{
   GP1:
	UF : 1, UT : 1,		CONFIG : 'N U T, 0, 0, 1',
	X =  31.000  mm,	Y =  52.000  mm,	Z =   15.000 mm,
	W =180.000 deg,	P =   0.000 deg,	R =    90.000 deg
};
P[3020]{
   GP1:
	UF : 1, UT : 1,		CONFIG : 'N U T, 0, 0, 1',
	X =  31.000  mm,	Y =  52.000  mm,	Z =   0.600 mm,
	W =180.000 deg,	P =   0.000 deg,	R =    90.000 deg
};
P[3021]{
   GP1:
	UF : 1, UT : 1,		CONFIG : 'N U T, 0, 0, 1',
	X =  31.000  mm,	Y =  52.000  mm,	Z =   15.000 mm,
	W =180.000 deg,	P =   0.000 deg,	R =    90.000 deg
};
P[3022]{
   GP1:
	UF : 1, UT : 1,		CONFIG : 'N U T, 0, 0, 1',
	X =  34.000  mm,	Y =  52.000  mm,	Z =   15.000 mm,
	W =180.000 deg,	P =   0.000 deg,	R =    90.000 deg
};
P[3023]{
   GP1:
	UF : 1, UT : 1,		CONFIG : 'N U T, 0, 0, 1',
	X =  34.000  mm,	Y =  52.000  mm,	Z =   0.600 mm,
	W =180.000 deg,	P =   0.000 deg,	R =    90.000 deg
};
P[3024]{
   GP1:
	UF : 1, UT : 1,		CONFIG : 'N U T, 0, 0, 1',
	X =  34.000  mm,	Y =  52.000  mm,	Z =   15.000 mm,
	W =180.000 deg,	P =   0.000 deg,	R =    90.000 deg
};
P[3025]{
   GP1:
	UF : 1, UT : 1,		CONFIG : 'N U T, 0, 0, 1',
	X =  37.000  mm,	Y =  52.000  mm,	Z =   15.000 mm,
	W =180.000 deg,	P =   0.000 deg,	R =    90.000 deg
};
P[3026]{
   GP1:
	UF : 1, UT : 1,		CONFIG : 'N U T, 0, 0, 1',
	X =  37.000  mm,	Y =  52.000  mm,	Z =   0.600 mm,
	W =180.000 deg,	P =   0.000 deg,	R =    90.000 deg
};
P[3027]{
   GP1:
	UF : 1, UT : 1,		CONFIG : 'N U T, 0, 0, 1',
	X =  37.000  mm,	Y =  52.000  mm,	Z =   15.000 mm,
	W =180.000 deg,	P =   0.000 deg,	R =    90.000 deg
};
P[3028]{
   GP1:
	UF : 1, UT : 1,		CONFIG : 'N U T, 0, 0, 1',
	X =  40.000  mm,	Y =  52.000  mm,	Z =   15.000 mm,
	W =180.000 deg,	P =   0.000 deg,	R =    90.000 deg
};
P[3029]{
   GP1:
	UF : 1, UT : 1,		CONFIG : 'N U T, 0, 0, 1',
	X =  40.000  mm,	Y =  52.000  mm,	Z =   0.600 mm,
	W =180.000 deg,	P =   0.000 deg,	R =    90.000 deg
};
P[3030]{
   GP1:
	UF : 1, UT : 1,		CONFIG : 'N U T, 0, 0, 1',
	X =  40.000  mm,	Y =  52.000  mm,	Z =   15.000 mm,
	W =180.000 deg,	P =   0.000 deg,	R =    90.000 deg
};
P[3031]{
   GP1:
	UF : 1, UT : 1,		CONFIG : 'N U T, 0, 0, 1',
	X =  43.000  mm,	Y =  52.000  mm,	Z =   15.000 mm,
	W =180.000 deg,	P =   0.000 deg,	R =    90.000 deg
};
P[3032]{
   GP1:
	UF : 1, UT : 1,		CONFIG : 'N U T, 0, 0, 1',
	X =  43.000  mm,	Y =  52.000  mm,	Z =   0.600 mm,
	W =180.000 deg,	P =   0.000 deg,	R =    90.000 deg
};
P[3033]{
   GP1:
	UF : 1, UT : 1,		CONFIG : 'N U T, 0, 0, 1',
	X =  43.000  mm,	Y =  52.000  mm,	Z =   15.000 mm,
	W =180.000 deg,	P =   0.000 deg,	R =    90.000 deg
};
P[3034]{
   GP1:
	UF : 1, UT : 1,		CONFIG : 'N U T, 0, 0, 1',
	X =  46.000  mm,	Y =  52.000  mm,	Z =   15.000 mm,
	W =180.000 deg,	P =   0.000 deg,	R =    90.000 deg
};
P[3035]{
   GP1:
	UF : 1, UT : 1,		CONFIG : 'N U T, 0, 0, 1',
	X =  46.000  mm,	Y =  52.000  mm,	Z =   0.600 mm,
	W =180.000 deg,	P =   0.000 deg,	R =    90.000 deg
};
P[3036]{
   GP1:
	UF : 1, UT : 1,		CONFIG : 'N U T, 0, 0, 1',
	X =  46.000  mm,	Y =  52.000  mm,	Z =   15.000 mm,
	W =180.000 deg,	P =   0.000 deg,	R =    90.000 deg
};
P[3037]{
   GP1:
	UF : 1, UT : 1,		CONFIG : 'N U T, 0, 0, 1',
	X =  49.000  mm,	Y =  52.000  mm,	Z =   15.000 mm,
	W =180.000 deg,	P =   0.000 deg,	R =    90.000 deg
};
P[3038]{
   GP1:
	UF : 1, UT : 1,		CONFIG : 'N U T, 0, 0, 1',
	X =  49.000  mm,	Y =  52.000  mm,	Z =   0.600 mm,
	W =180.000 deg,	P =   0.000 deg,	R =    90.000 deg
};
P[3039]{
   GP1:
	UF : 1, UT : 1,		CONFIG : 'N U T, 0, 0, 1',
	X =  49.000  mm,	Y =  52.000  mm,	Z =   15.000 mm,
	W =180.000 deg,	P =   0.000 deg,	R =    90.000 deg
};
P[3040]{
   GP1:
	UF : 1, UT : 1,		CONFIG : 'N U T, 0, 0, 1',
	X =  52.000  mm,	Y =  52.000  mm,	Z =   15.000 mm,
	W =180.000 deg,	P =   0.000 deg,	R =    90.000 deg
};
P[3041]{
   GP1:
	UF : 1, UT : 1,		CONFIG : 'N U T, 0, 0, 1',
	X =  52.000  mm,	Y =  52.000  mm,	Z =   0.600 mm,
	W =180.000 deg,	P =   0.000 deg,	R =    90.000 deg
};
P[3042]{
   GP1:
	UF : 1, UT : 1,		CONFIG : 'N U T, 0, 0, 1',
	X =  52.000  mm,	Y =  52.000  mm,	Z =   15.000 mm,
	W =180.000 deg,	P =   0.000 deg,	R =    90.000 deg
};
P[3043]{
   GP1:
	UF : 1, UT : 1,		CONFIG : 'N U T, 0, 0, 1',
	X =  55.000  mm,	Y =  52.000  mm,	Z =   15.000 mm,
	W =180.000 deg,	P =   0.000 deg,	R =    90.000 deg
};
P[3044]{
   GP1:
	UF : 1, UT : 1,		CONFIG : 'N U T, 0, 0, 1',
	X =  55.000  mm,	Y =  52.000  mm,	Z =   0.600 mm,
	W =180.000 deg,	P =   0.000 deg,	R =    90.000 deg
};
P[3045]{
   GP1:
	UF : 1, UT : 1,		CONFIG : 'N U T, 0, 0, 1',
	X =  55.000  mm,	Y =  52.000  mm,	Z =   15.000 mm,
	W =180.000 deg,	P =   0.000 deg,	R =    90.000 deg
};
P[3046]{
   GP1:
	UF : 1, UT : 1,		CONFIG : 'N U T, 0, 0, 1',
	X =  58.000  mm,	Y =  52.000  mm,	Z =   15.000 mm,
	W =180.000 deg,	P =   0.000 deg,	R =    90.000 deg
};
P[3047]{
   GP1:
	UF : 1, UT : 1,		CONFIG : 'N U T, 0, 0, 1',
	X =  58.000  mm,	Y =  52.000  mm,	Z =   0.600 mm,
	W =180.000 deg,	P =   0.000 deg,	R =    90.000 deg
};
P[3048]{
   GP1:
	UF : 1, UT : 1,		CONFIG : 'N U T, 0, 0, 1',
	X =  58.000  mm,	Y =  52.000  mm,	Z =   15.000 mm,
	W =180.000 deg,	P =   0.000 deg,	R =    90.000 deg
};
P[3049]{
   GP1:
	UF : 1, UT : 1,		CONFIG : 'N U T, 0, 0, 1',
	X =  61.000  mm,	Y =  52.000  mm,	Z =   15.000 mm,
	W =180.000 deg,	P =   0.000 deg,	R =    90.000 deg
};
P[3050]{
   GP1:
	UF : 1, UT : 1,		CONFIG : 'N U T, 0, 0, 1',
	X =  61.000  mm,	Y =  52.000  mm,	Z =   0.600 mm,
	W =180.000 deg,	P =   0.000 deg,	R =    90.000 deg
};
P[3051]{
   GP1:
	UF : 1, UT : 1,		CONFIG : 'N U T, 0, 0, 1',
	X =  61.000  mm,	Y =  52.000  mm,	Z =   15.000 mm,
	W =180.000 deg,	P =   0.000 deg,	R =    90.000 deg
};
P[3061]{
   GP1:
	UF : 1, UT : 1,		CONFIG : 'N U T, 0, 0, 1',
	X =  73.000  mm,	Y =  52.000  mm,	Z =   15.000 mm,
	W =180.000 deg,	P =   0.000 deg,	R =    90.000 deg
};
P[3062]{
   GP1:
	UF : 1, UT : 1,		CONFIG : 'N U T, 0, 0, 1',
	X =  73.000  mm,	Y =  52.000  mm,	Z =   0.600 mm,
	W =180.000 deg,	P =   0.000 deg,	R =    90.000 deg
};
P[3063]{
   GP1:
	UF : 1, UT : 1,		CONFIG : 'N U T, 0, 0, 1',
	X =  73.000  mm,	Y =  52.000  mm,	Z =   15.000 mm,
	W =180.000 deg,	P =   0.000 deg,	R =    90.000 deg
};
P[3064]{
   GP1:
	UF : 1, UT : 1,		CONFIG : 'N U T, 0, 0, 1',
	X =  76.000  mm,	Y =  52.000  mm,	Z =   15.000 mm,
	W =180.000 deg,	P =   0.000 deg,	R =    90.000 deg
};
P[3065]{
   GP1:
	UF : 1, UT : 1,		CONFIG : 'N U T, 0, 0, 1',
	X =  76.000  mm,	Y =  52.000  mm,	Z =   0.600 mm,
	W =180.000 deg,	P =   0.000 deg,	R =    90.000 deg
};
P[3066]{
   GP1:
	UF : 1, UT : 1,		CONFIG : 'N U T, 0, 0, 1',
	X =  76.000  mm,	Y =  52.000  mm,	Z =   15.000 mm,
	W =180.000 deg,	P =   0.000 deg,	R =    90.000 deg
};
P[3067]{
   GP1:
	UF : 1, UT : 1,		CONFIG : 'N U T, 0, 0, 1',
	X =  79.000  mm,	Y =  52.000  mm,	Z =   15.000 mm,
	W =180.000 deg,	P =   0.000 deg,	R =    90.000 deg
};
P[3068]{
   GP1:
	UF : 1, UT : 1,		CONFIG : 'N U T, 0, 0, 1',
	X =  79.000  mm,	Y =  52.000  mm,	Z =   0.600 mm,
	W =180.000 deg,	P =   0.000 deg,	R =    90.000 deg
};
P[3069]{
   GP1:
	UF : 1, UT : 1,		CONFIG : 'N U T, 0, 0, 1',
	X =  79.000  mm,	Y =  52.000  mm,	Z =   15.000 mm,
	W =180.000 deg,	P =   0.000 deg,	R =    90.000 deg
};
P[3076]{
   GP1:
	UF : 1, UT : 1,		CONFIG : 'N U T, 0, 0, 1',
	X =  88.000  mm,	Y =  52.000  mm,	Z =   15.000 mm,
	W =180.000 deg,	P =   0.000 deg,	R =    90.000 deg
};
P[3077]{
   GP1:
	UF : 1, UT : 1,		CONFIG : 'N U T, 0, 0, 1',
	X =  88.000  mm,	Y =  52.000  mm,	Z =   0.600 mm,
	W =180.000 deg,	P =   0.000 deg,	R =    90.000 deg
};
P[3078]{
   GP1:
	UF : 1, UT : 1,		CONFIG : 'N U T, 0, 0, 1',
	X =  88.000  mm,	Y =  52.000  mm,	Z =   15.000 mm,
	W =180.000 deg,	P =   0.000 deg,	R =    90.000 deg
};
P[3079]{
   GP1:
	UF : 1, UT : 1,		CONFIG : 'N U T, 0, 0, 1',
	X =  91.000  mm,	Y =  52.000  mm,	Z =   15.000 mm,
	W =180.000 deg,	P =   0.000 deg,	R =    90.000 deg
};
P[3080]{
   GP1:
	UF : 1, UT : 1,		CONFIG : 'N U T, 0, 0, 1',
	X =  91.000  mm,	Y =  52.000  mm,	Z =   0.600 mm,
	W =180.000 deg,	P =   0.000 deg,	R =    90.000 deg
};
P[3081]{
   GP1:
	UF : 1, UT : 1,		CONFIG : 'N U T, 0, 0, 1',
	X =  91.000  mm,	Y =  52.000  mm,	Z =   15.000 mm,
	W =180.000 deg,	P =   0.000 deg,	R =    90.000 deg
};
P[3082]{
   GP1:
	UF : 1, UT : 1,		CONFIG : 'N U T, 0, 0, 1',
	X =  94.000  mm,	Y =  52.000  mm,	Z =   15.000 mm,
	W =180.000 deg,	P =   0.000 deg,	R =    90.000 deg
};
P[3083]{
   GP1:
	UF : 1, UT : 1,		CONFIG : 'N U T, 0, 0, 1',
	X =  94.000  mm,	Y =  52.000  mm,	Z =   0.600 mm,
	W =180.000 deg,	P =   0.000 deg,	R =    90.000 deg
};
P[3084]{
   GP1:
	UF : 1, UT : 1,		CONFIG : 'N U T, 0, 0, 1',
	X =  94.000  mm,	Y =  52.000  mm,	Z =   15.000 mm,
	W =180.000 deg,	P =   0.000 deg,	R =    90.000 deg
};
P[3085]{
   GP1:
	UF : 1, UT : 1,		CONFIG : 'N U T, 0, 0, 1',
	X =  97.000  mm,	Y =  52.000  mm,	Z =   15.000 mm,
	W =180.000 deg,	P =   0.000 deg,	R =    90.000 deg
};
P[3086]{
   GP1:
	UF : 1, UT : 1,		CONFIG : 'N U T, 0, 0, 1',
	X =  97.000  mm,	Y =  52.000  mm,	Z =   0.600 mm,
	W =180.000 deg,	P =   0.000 deg,	R =    90.000 deg
};
P[3087]{
   GP1:
	UF : 1, UT : 1,		CONFIG : 'N U T, 0, 0, 1',
	X =  97.000  mm,	Y =  52.000  mm,	Z =   15.000 mm,
	W =180.000 deg,	P =   0.000 deg,	R =    90.000 deg
};
P[3088]{
   GP1:
	UF : 1, UT : 1,		CONFIG : 'N U T, 0, 0, 1',
	X =  100.000  mm,	Y =  52.000  mm,	Z =   15.000 mm,
	W =180.000 deg,	P =   0.000 deg,	R =    90.000 deg
};
P[3089]{
   GP1:
	UF : 1, UT : 1,		CONFIG : 'N U T, 0, 0, 1',
	X =  100.000  mm,	Y =  52.000  mm,	Z =   0.600 mm,
	W =180.000 deg,	P =   0.000 deg,	R =    90.000 deg
};
P[3090]{
   GP1:
	UF : 1, UT : 1,		CONFIG : 'N U T, 0, 0, 1',
	X =  100.000  mm,	Y =  52.000  mm,	Z =   15.000 mm,
	W =180.000 deg,	P =   0.000 deg,	R =    90.000 deg
};
P[3091]{
   GP1:
	UF : 1, UT : 1,		CONFIG : 'N U T, 0, 0, 1',
	X =  103.000  mm,	Y =  52.000  mm,	Z =   15.000 mm,
	W =180.000 deg,	P =   0.000 deg,	R =    90.000 deg
};
P[3092]{
   GP1:
	UF : 1, UT : 1,		CONFIG : 'N U T, 0, 0, 1',
	X =  103.000  mm,	Y =  52.000  mm,	Z =   0.600 mm,
	W =180.000 deg,	P =   0.000 deg,	R =    90.000 deg
};
P[3093]{
   GP1:
	UF : 1, UT : 1,		CONFIG : 'N U T, 0, 0, 1',
	X =  103.000  mm,	Y =  52.000  mm,	Z =   15.000 mm,
	W =180.000 deg,	P =   0.000 deg,	R =    90.000 deg
};
P[3094]{
   GP1:
	UF : 1, UT : 1,		CONFIG : 'N U T, 0, 0, 1',
	X =  106.000  mm,	Y =  52.000  mm,	Z =   15.000 mm,
	W =180.000 deg,	P =   0.000 deg,	R =    90.000 deg
};
P[3095]{
   GP1:
	UF : 1, UT : 1,		CONFIG : 'N U T, 0, 0, 1',
	X =  106.000  mm,	Y =  52.000  mm,	Z =   0.600 mm,
	W =180.000 deg,	P =   0.000 deg,	R =    90.000 deg
};
P[3096]{
   GP1:
	UF : 1, UT : 1,		CONFIG : 'N U T, 0, 0, 1',
	X =  106.000  mm,	Y =  52.000  mm,	Z =   15.000 mm,
	W =180.000 deg,	P =   0.000 deg,	R =    90.000 deg
};
P[3097]{
   GP1:
	UF : 1, UT : 1,		CONFIG : 'N U T, 0, 0, 1',
	X =  109.000  mm,	Y =  52.000  mm,	Z =   15.000 mm,
	W =180.000 deg,	P =   0.000 deg,	R =    90.000 deg
};
P[3098]{
   GP1:
	UF : 1, UT : 1,		CONFIG : 'N U T, 0, 0, 1',
	X =  109.000  mm,	Y =  52.000  mm,	Z =   0.600 mm,
	W =180.000 deg,	P =   0.000 deg,	R =    90.000 deg
};
P[3099]{
   GP1:
	UF : 1, UT : 1,		CONFIG : 'N U T, 0, 0, 1',
	X =  109.000  mm,	Y =  52.000  mm,	Z =   15.000 mm,
	W =180.000 deg,	P =   0.000 deg,	R =    90.000 deg
};
P[3100]{
   GP1:
	UF : 1, UT : 1,		CONFIG : 'N U T, 0, 0, 1',
	X =  112.000  mm,	Y =  52.000  mm,	Z =   15.000 mm,
	W =180.000 deg,	P =   0.000 deg,	R =    90.000 deg
};
P[3101]{
   GP1:
	UF : 1, UT : 1,		CONFIG : 'N U T, 0, 0, 1',
	X =  112.000  mm,	Y =  52.000  mm,	Z =   0.600 mm,
	W =180.000 deg,	P =   0.000 deg,	R =    90.000 deg
};
P[3102]{
   GP1:
	UF : 1, UT : 1,		CONFIG : 'N U T, 0, 0, 1',
	X =  112.000  mm,	Y =  52.000  mm,	Z =   15.000 mm,
	W =180.000 deg,	P =   0.000 deg,	R =    90.000 deg
};
P[3106]{
   GP1:
	UF : 1, UT : 1,		CONFIG : 'N U T, 0, 0, 1',
	X =  127.000  mm,	Y =  52.000  mm,	Z =   15.000 mm,
	W =180.000 deg,	P =   0.000 deg,	R =    90.000 deg
};
P[3107]{
   GP1:
	UF : 1, UT : 1,		CONFIG : 'N U T, 0, 0, 1',
	X =  127.000  mm,	Y =  52.000  mm,	Z =   0.600 mm,
	W =180.000 deg,	P =   0.000 deg,	R =    90.000 deg
};
P[3108]{
   GP1:
	UF : 1, UT : 1,		CONFIG : 'N U T, 0, 0, 1',
	X =  127.000  mm,	Y =  52.000  mm,	Z =   15.000 mm,
	W =180.000 deg,	P =   0.000 deg,	R =    90.000 deg
};
P[3112]{
   GP1:
	UF : 1, UT : 1,		CONFIG : 'N U T, 0, 0, 1',
	X =  133.000  mm,	Y =  52.000  mm,	Z =   15.000 mm,
	W =180.000 deg,	P =   0.000 deg,	R =    90.000 deg
};
P[3113]{
   GP1:
	UF : 1, UT : 1,		CONFIG : 'N U T, 0, 0, 1',
	X =  133.000  mm,	Y =  52.000  mm,	Z =   0.600 mm,
	W =180.000 deg,	P =   0.000 deg,	R =    90.000 deg
};
P[3114]{
   GP1:
	UF : 1, UT : 1,		CONFIG : 'N U T, 0, 0, 1',
	X =  133.000  mm,	Y =  52.000  mm,	Z =   15.000 mm,
	W =180.000 deg,	P =   0.000 deg,	R =    90.000 deg
};
P[3115]{
   GP1:
	UF : 1, UT : 1,		CONFIG : 'N U T, 0, 0, 1',
	X =  136.000  mm,	Y =  52.000  mm,	Z =   15.000 mm,
	W =180.000 deg,	P =   0.000 deg,	R =    90.000 deg
};
P[3116]{
   GP1:
	UF : 1, UT : 1,		CONFIG : 'N U T, 0, 0, 1',
	X =  136.000  mm,	Y =  52.000  mm,	Z =   0.600 mm,
	W =180.000 deg,	P =   0.000 deg,	R =    90.000 deg
};
P[3117]{
   GP1:
	UF : 1, UT : 1,		CONFIG : 'N U T, 0, 0, 1',
	X =  136.000  mm,	Y =  52.000  mm,	Z =   15.000 mm,
	W =180.000 deg,	P =   0.000 deg,	R =    90.000 deg
};
P[3118]{
   GP1:
	UF : 1, UT : 1,		CONFIG : 'N U T, 0, 0, 1',
	X =  139.000  mm,	Y =  52.000  mm,	Z =   15.000 mm,
	W =180.000 deg,	P =   0.000 deg,	R =    90.000 deg
};
P[3119]{
   GP1:
	UF : 1, UT : 1,		CONFIG : 'N U T, 0, 0, 1',
	X =  139.000  mm,	Y =  52.000  mm,	Z =   0.600 mm,
	W =180.000 deg,	P =   0.000 deg,	R =    90.000 deg
};
P[3120]{
   GP1:
	UF : 1, UT : 1,		CONFIG : 'N U T, 0, 0, 1',
	X =  139.000  mm,	Y =  52.000  mm,	Z =   15.000 mm,
	W =180.000 deg,	P =   0.000 deg,	R =    90.000 deg
};
P[3133]{
   GP1:
	UF : 1, UT : 1,		CONFIG : 'N U T, 0, 0, 1',
	X =  175.000  mm,	Y =  52.000  mm,	Z =   15.000 mm,
	W =180.000 deg,	P =   0.000 deg,	R =    90.000 deg
};
P[3134]{
   GP1:
	UF : 1, UT : 1,		CONFIG : 'N U T, 0, 0, 1',
	X =  175.000  mm,	Y =  52.000  mm,	Z =   0.600 mm,
	W =180.000 deg,	P =   0.000 deg,	R =    90.000 deg
};
P[3135]{
   GP1:
	UF : 1, UT : 1,		CONFIG : 'N U T, 0, 0, 1',
	X =  175.000  mm,	Y =  52.000  mm,	Z =   15.000 mm,
	W =180.000 deg,	P =   0.000 deg,	R =    90.000 deg
};
P[3136]{
   GP1:
	UF : 1, UT : 1,		CONFIG : 'N U T, 0, 0, 1',
	X =  178.000  mm,	Y =  52.000  mm,	Z =   15.000 mm,
	W =180.000 deg,	P =   0.000 deg,	R =    90.000 deg
};
P[3137]{
   GP1:
	UF : 1, UT : 1,		CONFIG : 'N U T, 0, 0, 1',
	X =  178.000  mm,	Y =  52.000  mm,	Z =   0.600 mm,
	W =180.000 deg,	P =   0.000 deg,	R =    90.000 deg
};
P[3138]{
   GP1:
	UF : 1, UT : 1,		CONFIG : 'N U T, 0, 0, 1',
	X =  178.000  mm,	Y =  52.000  mm,	Z =   15.000 mm,
	W =180.000 deg,	P =   0.000 deg,	R =    90.000 deg
};
P[3139]{
   GP1:
	UF : 1, UT : 1,		CONFIG : 'N U T, 0, 0, 1',
	X =  1.000  mm,	Y =  55.000  mm,	Z =   15.000 mm,
	W =180.000 deg,	P =   0.000 deg,	R =    90.000 deg
};
P[3140]{
   GP1:
	UF : 1, UT : 1,		CONFIG : 'N U T, 0, 0, 1',
	X =  1.000  mm,	Y =  55.000  mm,	Z =   0.600 mm,
	W =180.000 deg,	P =   0.000 deg,	R =    90.000 deg
};
P[3141]{
   GP1:
	UF : 1, UT : 1,		CONFIG : 'N U T, 0, 0, 1',
	X =  1.000  mm,	Y =  55.000  mm,	Z =   15.000 mm,
	W =180.000 deg,	P =   0.000 deg,	R =    90.000 deg
};
P[3142]{
   GP1:
	UF : 1, UT : 1,		CONFIG : 'N U T, 0, 0, 1',
	X =  4.000  mm,	Y =  55.000  mm,	Z =   15.000 mm,
	W =180.000 deg,	P =   0.000 deg,	R =    90.000 deg
};
P[3143]{
   GP1:
	UF : 1, UT : 1,		CONFIG : 'N U T, 0, 0, 1',
	X =  4.000  mm,	Y =  55.000  mm,	Z =   0.600 mm,
	W =180.000 deg,	P =   0.000 deg,	R =    90.000 deg
};
P[3144]{
   GP1:
	UF : 1, UT : 1,		CONFIG : 'N U T, 0, 0, 1',
	X =  4.000  mm,	Y =  55.000  mm,	Z =   15.000 mm,
	W =180.000 deg,	P =   0.000 deg,	R =    90.000 deg
};
P[3145]{
   GP1:
	UF : 1, UT : 1,		CONFIG : 'N U T, 0, 0, 1',
	X =  7.000  mm,	Y =  55.000  mm,	Z =   15.000 mm,
	W =180.000 deg,	P =   0.000 deg,	R =    90.000 deg
};
P[3146]{
   GP1:
	UF : 1, UT : 1,		CONFIG : 'N U T, 0, 0, 1',
	X =  7.000  mm,	Y =  55.000  mm,	Z =   0.600 mm,
	W =180.000 deg,	P =   0.000 deg,	R =    90.000 deg
};
P[3147]{
   GP1:
	UF : 1, UT : 1,		CONFIG : 'N U T, 0, 0, 1',
	X =  7.000  mm,	Y =  55.000  mm,	Z =   15.000 mm,
	W =180.000 deg,	P =   0.000 deg,	R =    90.000 deg
};
P[3148]{
   GP1:
	UF : 1, UT : 1,		CONFIG : 'N U T, 0, 0, 1',
	X =  10.000  mm,	Y =  55.000  mm,	Z =   15.000 mm,
	W =180.000 deg,	P =   0.000 deg,	R =    90.000 deg
};
P[3149]{
   GP1:
	UF : 1, UT : 1,		CONFIG : 'N U T, 0, 0, 1',
	X =  10.000  mm,	Y =  55.000  mm,	Z =   0.600 mm,
	W =180.000 deg,	P =   0.000 deg,	R =    90.000 deg
};
P[3150]{
   GP1:
	UF : 1, UT : 1,		CONFIG : 'N U T, 0, 0, 1',
	X =  10.000  mm,	Y =  55.000  mm,	Z =   15.000 mm,
	W =180.000 deg,	P =   0.000 deg,	R =    90.000 deg
};
P[3151]{
   GP1:
	UF : 1, UT : 1,		CONFIG : 'N U T, 0, 0, 1',
	X =  13.000  mm,	Y =  55.000  mm,	Z =   15.000 mm,
	W =180.000 deg,	P =   0.000 deg,	R =    90.000 deg
};
P[3152]{
   GP1:
	UF : 1, UT : 1,		CONFIG : 'N U T, 0, 0, 1',
	X =  13.000  mm,	Y =  55.000  mm,	Z =   0.600 mm,
	W =180.000 deg,	P =   0.000 deg,	R =    90.000 deg
};
P[3153]{
   GP1:
	UF : 1, UT : 1,		CONFIG : 'N U T, 0, 0, 1',
	X =  13.000  mm,	Y =  55.000  mm,	Z =   15.000 mm,
	W =180.000 deg,	P =   0.000 deg,	R =    90.000 deg
};
P[3154]{
   GP1:
	UF : 1, UT : 1,		CONFIG : 'N U T, 0, 0, 1',
	X =  16.000  mm,	Y =  55.000  mm,	Z =   15.000 mm,
	W =180.000 deg,	P =   0.000 deg,	R =    90.000 deg
};
P[3155]{
   GP1:
	UF : 1, UT : 1,		CONFIG : 'N U T, 0, 0, 1',
	X =  16.000  mm,	Y =  55.000  mm,	Z =   0.600 mm,
	W =180.000 deg,	P =   0.000 deg,	R =    90.000 deg
};
P[3156]{
   GP1:
	UF : 1, UT : 1,		CONFIG : 'N U T, 0, 0, 1',
	X =  16.000  mm,	Y =  55.000  mm,	Z =   15.000 mm,
	W =180.000 deg,	P =   0.000 deg,	R =    90.000 deg
};
P[3157]{
   GP1:
	UF : 1, UT : 1,		CONFIG : 'N U T, 0, 0, 1',
	X =  19.000  mm,	Y =  55.000  mm,	Z =   15.000 mm,
	W =180.000 deg,	P =   0.000 deg,	R =    90.000 deg
};
P[3158]{
   GP1:
	UF : 1, UT : 1,		CONFIG : 'N U T, 0, 0, 1',
	X =  19.000  mm,	Y =  55.000  mm,	Z =   0.600 mm,
	W =180.000 deg,	P =   0.000 deg,	R =    90.000 deg
};
P[3159]{
   GP1:
	UF : 1, UT : 1,		CONFIG : 'N U T, 0, 0, 1',
	X =  19.000  mm,	Y =  55.000  mm,	Z =   15.000 mm,
	W =180.000 deg,	P =   0.000 deg,	R =    90.000 deg
};
P[3160]{
   GP1:
	UF : 1, UT : 1,		CONFIG : 'N U T, 0, 0, 1',
	X =  25.000  mm,	Y =  55.000  mm,	Z =   15.000 mm,
	W =180.000 deg,	P =   0.000 deg,	R =    90.000 deg
};
P[3161]{
   GP1:
	UF : 1, UT : 1,		CONFIG : 'N U T, 0, 0, 1',
	X =  25.000  mm,	Y =  55.000  mm,	Z =   0.600 mm,
	W =180.000 deg,	P =   0.000 deg,	R =    90.000 deg
};
P[3162]{
   GP1:
	UF : 1, UT : 1,		CONFIG : 'N U T, 0, 0, 1',
	X =  25.000  mm,	Y =  55.000  mm,	Z =   15.000 mm,
	W =180.000 deg,	P =   0.000 deg,	R =    90.000 deg
};
P[3163]{
   GP1:
	UF : 1, UT : 1,		CONFIG : 'N U T, 0, 0, 1',
	X =  28.000  mm,	Y =  55.000  mm,	Z =   15.000 mm,
	W =180.000 deg,	P =   0.000 deg,	R =    90.000 deg
};
P[3164]{
   GP1:
	UF : 1, UT : 1,		CONFIG : 'N U T, 0, 0, 1',
	X =  28.000  mm,	Y =  55.000  mm,	Z =   0.600 mm,
	W =180.000 deg,	P =   0.000 deg,	R =    90.000 deg
};
P[3165]{
   GP1:
	UF : 1, UT : 1,		CONFIG : 'N U T, 0, 0, 1',
	X =  28.000  mm,	Y =  55.000  mm,	Z =   15.000 mm,
	W =180.000 deg,	P =   0.000 deg,	R =    90.000 deg
};
P[3166]{
   GP1:
	UF : 1, UT : 1,		CONFIG : 'N U T, 0, 0, 1',
	X =  31.000  mm,	Y =  55.000  mm,	Z =   15.000 mm,
	W =180.000 deg,	P =   0.000 deg,	R =    90.000 deg
};
P[3167]{
   GP1:
	UF : 1, UT : 1,		CONFIG : 'N U T, 0, 0, 1',
	X =  31.000  mm,	Y =  55.000  mm,	Z =   0.600 mm,
	W =180.000 deg,	P =   0.000 deg,	R =    90.000 deg
};
P[3168]{
   GP1:
	UF : 1, UT : 1,		CONFIG : 'N U T, 0, 0, 1',
	X =  31.000  mm,	Y =  55.000  mm,	Z =   15.000 mm,
	W =180.000 deg,	P =   0.000 deg,	R =    90.000 deg
};
P[3169]{
   GP1:
	UF : 1, UT : 1,		CONFIG : 'N U T, 0, 0, 1',
	X =  34.000  mm,	Y =  55.000  mm,	Z =   15.000 mm,
	W =180.000 deg,	P =   0.000 deg,	R =    90.000 deg
};
P[3170]{
   GP1:
	UF : 1, UT : 1,		CONFIG : 'N U T, 0, 0, 1',
	X =  34.000  mm,	Y =  55.000  mm,	Z =   0.600 mm,
	W =180.000 deg,	P =   0.000 deg,	R =    90.000 deg
};
P[3171]{
   GP1:
	UF : 1, UT : 1,		CONFIG : 'N U T, 0, 0, 1',
	X =  34.000  mm,	Y =  55.000  mm,	Z =   15.000 mm,
	W =180.000 deg,	P =   0.000 deg,	R =    90.000 deg
};
P[3172]{
   GP1:
	UF : 1, UT : 1,		CONFIG : 'N U T, 0, 0, 1',
	X =  37.000  mm,	Y =  55.000  mm,	Z =   15.000 mm,
	W =180.000 deg,	P =   0.000 deg,	R =    90.000 deg
};
P[3173]{
   GP1:
	UF : 1, UT : 1,		CONFIG : 'N U T, 0, 0, 1',
	X =  37.000  mm,	Y =  55.000  mm,	Z =   0.600 mm,
	W =180.000 deg,	P =   0.000 deg,	R =    90.000 deg
};
P[3174]{
   GP1:
	UF : 1, UT : 1,		CONFIG : 'N U T, 0, 0, 1',
	X =  37.000  mm,	Y =  55.000  mm,	Z =   15.000 mm,
	W =180.000 deg,	P =   0.000 deg,	R =    90.000 deg
};
P[3175]{
   GP1:
	UF : 1, UT : 1,		CONFIG : 'N U T, 0, 0, 1',
	X =  40.000  mm,	Y =  55.000  mm,	Z =   15.000 mm,
	W =180.000 deg,	P =   0.000 deg,	R =    90.000 deg
};
P[3176]{
   GP1:
	UF : 1, UT : 1,		CONFIG : 'N U T, 0, 0, 1',
	X =  40.000  mm,	Y =  55.000  mm,	Z =   0.600 mm,
	W =180.000 deg,	P =   0.000 deg,	R =    90.000 deg
};
P[3177]{
   GP1:
	UF : 1, UT : 1,		CONFIG : 'N U T, 0, 0, 1',
	X =  40.000  mm,	Y =  55.000  mm,	Z =   15.000 mm,
	W =180.000 deg,	P =   0.000 deg,	R =    90.000 deg
};
P[3178]{
   GP1:
	UF : 1, UT : 1,		CONFIG : 'N U T, 0, 0, 1',
	X =  43.000  mm,	Y =  55.000  mm,	Z =   15.000 mm,
	W =180.000 deg,	P =   0.000 deg,	R =    90.000 deg
};
P[3179]{
   GP1:
	UF : 1, UT : 1,		CONFIG : 'N U T, 0, 0, 1',
	X =  43.000  mm,	Y =  55.000  mm,	Z =   0.600 mm,
	W =180.000 deg,	P =   0.000 deg,	R =    90.000 deg
};
P[3180]{
   GP1:
	UF : 1, UT : 1,		CONFIG : 'N U T, 0, 0, 1',
	X =  43.000  mm,	Y =  55.000  mm,	Z =   15.000 mm,
	W =180.000 deg,	P =   0.000 deg,	R =    90.000 deg
};
P[3181]{
   GP1:
	UF : 1, UT : 1,		CONFIG : 'N U T, 0, 0, 1',
	X =  46.000  mm,	Y =  55.000  mm,	Z =   15.000 mm,
	W =180.000 deg,	P =   0.000 deg,	R =    90.000 deg
};
P[3182]{
   GP1:
	UF : 1, UT : 1,		CONFIG : 'N U T, 0, 0, 1',
	X =  46.000  mm,	Y =  55.000  mm,	Z =   0.600 mm,
	W =180.000 deg,	P =   0.000 deg,	R =    90.000 deg
};
P[3183]{
   GP1:
	UF : 1, UT : 1,		CONFIG : 'N U T, 0, 0, 1',
	X =  46.000  mm,	Y =  55.000  mm,	Z =   15.000 mm,
	W =180.000 deg,	P =   0.000 deg,	R =    90.000 deg
};
P[3184]{
   GP1:
	UF : 1, UT : 1,		CONFIG : 'N U T, 0, 0, 1',
	X =  49.000  mm,	Y =  55.000  mm,	Z =   15.000 mm,
	W =180.000 deg,	P =   0.000 deg,	R =    90.000 deg
};
P[3185]{
   GP1:
	UF : 1, UT : 1,		CONFIG : 'N U T, 0, 0, 1',
	X =  49.000  mm,	Y =  55.000  mm,	Z =   0.600 mm,
	W =180.000 deg,	P =   0.000 deg,	R =    90.000 deg
};
P[3186]{
   GP1:
	UF : 1, UT : 1,		CONFIG : 'N U T, 0, 0, 1',
	X =  49.000  mm,	Y =  55.000  mm,	Z =   15.000 mm,
	W =180.000 deg,	P =   0.000 deg,	R =    90.000 deg
};
P[3187]{
   GP1:
	UF : 1, UT : 1,		CONFIG : 'N U T, 0, 0, 1',
	X =  52.000  mm,	Y =  55.000  mm,	Z =   15.000 mm,
	W =180.000 deg,	P =   0.000 deg,	R =    90.000 deg
};
P[3188]{
   GP1:
	UF : 1, UT : 1,		CONFIG : 'N U T, 0, 0, 1',
	X =  52.000  mm,	Y =  55.000  mm,	Z =   0.600 mm,
	W =180.000 deg,	P =   0.000 deg,	R =    90.000 deg
};
P[3189]{
   GP1:
	UF : 1, UT : 1,		CONFIG : 'N U T, 0, 0, 1',
	X =  52.000  mm,	Y =  55.000  mm,	Z =   15.000 mm,
	W =180.000 deg,	P =   0.000 deg,	R =    90.000 deg
};
P[3190]{
   GP1:
	UF : 1, UT : 1,		CONFIG : 'N U T, 0, 0, 1',
	X =  55.000  mm,	Y =  55.000  mm,	Z =   15.000 mm,
	W =180.000 deg,	P =   0.000 deg,	R =    90.000 deg
};
P[3191]{
   GP1:
	UF : 1, UT : 1,		CONFIG : 'N U T, 0, 0, 1',
	X =  55.000  mm,	Y =  55.000  mm,	Z =   0.600 mm,
	W =180.000 deg,	P =   0.000 deg,	R =    90.000 deg
};
P[3192]{
   GP1:
	UF : 1, UT : 1,		CONFIG : 'N U T, 0, 0, 1',
	X =  55.000  mm,	Y =  55.000  mm,	Z =   15.000 mm,
	W =180.000 deg,	P =   0.000 deg,	R =    90.000 deg
};
P[3193]{
   GP1:
	UF : 1, UT : 1,		CONFIG : 'N U T, 0, 0, 1',
	X =  58.000  mm,	Y =  55.000  mm,	Z =   15.000 mm,
	W =180.000 deg,	P =   0.000 deg,	R =    90.000 deg
};
P[3194]{
   GP1:
	UF : 1, UT : 1,		CONFIG : 'N U T, 0, 0, 1',
	X =  58.000  mm,	Y =  55.000  mm,	Z =   0.600 mm,
	W =180.000 deg,	P =   0.000 deg,	R =    90.000 deg
};
P[3195]{
   GP1:
	UF : 1, UT : 1,		CONFIG : 'N U T, 0, 0, 1',
	X =  58.000  mm,	Y =  55.000  mm,	Z =   15.000 mm,
	W =180.000 deg,	P =   0.000 deg,	R =    90.000 deg
};
P[3196]{
   GP1:
	UF : 1, UT : 1,		CONFIG : 'N U T, 0, 0, 1',
	X =  61.000  mm,	Y =  55.000  mm,	Z =   15.000 mm,
	W =180.000 deg,	P =   0.000 deg,	R =    90.000 deg
};
P[3197]{
   GP1:
	UF : 1, UT : 1,		CONFIG : 'N U T, 0, 0, 1',
	X =  61.000  mm,	Y =  55.000  mm,	Z =   0.600 mm,
	W =180.000 deg,	P =   0.000 deg,	R =    90.000 deg
};
P[3198]{
   GP1:
	UF : 1, UT : 1,		CONFIG : 'N U T, 0, 0, 1',
	X =  61.000  mm,	Y =  55.000  mm,	Z =   15.000 mm,
	W =180.000 deg,	P =   0.000 deg,	R =    90.000 deg
};
P[3211]{
   GP1:
	UF : 1, UT : 1,		CONFIG : 'N U T, 0, 0, 1',
	X =  76.000  mm,	Y =  55.000  mm,	Z =   15.000 mm,
	W =180.000 deg,	P =   0.000 deg,	R =    90.000 deg
};
P[3212]{
   GP1:
	UF : 1, UT : 1,		CONFIG : 'N U T, 0, 0, 1',
	X =  76.000  mm,	Y =  55.000  mm,	Z =   0.600 mm,
	W =180.000 deg,	P =   0.000 deg,	R =    90.000 deg
};
P[3213]{
   GP1:
	UF : 1, UT : 1,		CONFIG : 'N U T, 0, 0, 1',
	X =  76.000  mm,	Y =  55.000  mm,	Z =   15.000 mm,
	W =180.000 deg,	P =   0.000 deg,	R =    90.000 deg
};
P[3214]{
   GP1:
	UF : 1, UT : 1,		CONFIG : 'N U T, 0, 0, 1',
	X =  79.000  mm,	Y =  55.000  mm,	Z =   15.000 mm,
	W =180.000 deg,	P =   0.000 deg,	R =    90.000 deg
};
P[3215]{
   GP1:
	UF : 1, UT : 1,		CONFIG : 'N U T, 0, 0, 1',
	X =  79.000  mm,	Y =  55.000  mm,	Z =   0.600 mm,
	W =180.000 deg,	P =   0.000 deg,	R =    90.000 deg
};
P[3216]{
   GP1:
	UF : 1, UT : 1,		CONFIG : 'N U T, 0, 0, 1',
	X =  79.000  mm,	Y =  55.000  mm,	Z =   15.000 mm,
	W =180.000 deg,	P =   0.000 deg,	R =    90.000 deg
};
P[3223]{
   GP1:
	UF : 1, UT : 1,		CONFIG : 'N U T, 0, 0, 1',
	X =  88.000  mm,	Y =  55.000  mm,	Z =   15.000 mm,
	W =180.000 deg,	P =   0.000 deg,	R =    90.000 deg
};
P[3224]{
   GP1:
	UF : 1, UT : 1,		CONFIG : 'N U T, 0, 0, 1',
	X =  88.000  mm,	Y =  55.000  mm,	Z =   0.600 mm,
	W =180.000 deg,	P =   0.000 deg,	R =    90.000 deg
};
P[3225]{
   GP1:
	UF : 1, UT : 1,		CONFIG : 'N U T, 0, 0, 1',
	X =  88.000  mm,	Y =  55.000  mm,	Z =   15.000 mm,
	W =180.000 deg,	P =   0.000 deg,	R =    90.000 deg
};
P[3226]{
   GP1:
	UF : 1, UT : 1,		CONFIG : 'N U T, 0, 0, 1',
	X =  91.000  mm,	Y =  55.000  mm,	Z =   15.000 mm,
	W =180.000 deg,	P =   0.000 deg,	R =    90.000 deg
};
P[3227]{
   GP1:
	UF : 1, UT : 1,		CONFIG : 'N U T, 0, 0, 1',
	X =  91.000  mm,	Y =  55.000  mm,	Z =   0.600 mm,
	W =180.000 deg,	P =   0.000 deg,	R =    90.000 deg
};
P[3228]{
   GP1:
	UF : 1, UT : 1,		CONFIG : 'N U T, 0, 0, 1',
	X =  91.000  mm,	Y =  55.000  mm,	Z =   15.000 mm,
	W =180.000 deg,	P =   0.000 deg,	R =    90.000 deg
};
P[3229]{
   GP1:
	UF : 1, UT : 1,		CONFIG : 'N U T, 0, 0, 1',
	X =  94.000  mm,	Y =  55.000  mm,	Z =   15.000 mm,
	W =180.000 deg,	P =   0.000 deg,	R =    90.000 deg
};
P[3230]{
   GP1:
	UF : 1, UT : 1,		CONFIG : 'N U T, 0, 0, 1',
	X =  94.000  mm,	Y =  55.000  mm,	Z =   0.600 mm,
	W =180.000 deg,	P =   0.000 deg,	R =    90.000 deg
};
P[3231]{
   GP1:
	UF : 1, UT : 1,		CONFIG : 'N U T, 0, 0, 1',
	X =  94.000  mm,	Y =  55.000  mm,	Z =   15.000 mm,
	W =180.000 deg,	P =   0.000 deg,	R =    90.000 deg
};
P[3232]{
   GP1:
	UF : 1, UT : 1,		CONFIG : 'N U T, 0, 0, 1',
	X =  97.000  mm,	Y =  55.000  mm,	Z =   15.000 mm,
	W =180.000 deg,	P =   0.000 deg,	R =    90.000 deg
};
P[3233]{
   GP1:
	UF : 1, UT : 1,		CONFIG : 'N U T, 0, 0, 1',
	X =  97.000  mm,	Y =  55.000  mm,	Z =   0.600 mm,
	W =180.000 deg,	P =   0.000 deg,	R =    90.000 deg
};
P[3234]{
   GP1:
	UF : 1, UT : 1,		CONFIG : 'N U T, 0, 0, 1',
	X =  97.000  mm,	Y =  55.000  mm,	Z =   15.000 mm,
	W =180.000 deg,	P =   0.000 deg,	R =    90.000 deg
};
P[3235]{
   GP1:
	UF : 1, UT : 1,		CONFIG : 'N U T, 0, 0, 1',
	X =  100.000  mm,	Y =  55.000  mm,	Z =   15.000 mm,
	W =180.000 deg,	P =   0.000 deg,	R =    90.000 deg
};
P[3236]{
   GP1:
	UF : 1, UT : 1,		CONFIG : 'N U T, 0, 0, 1',
	X =  100.000  mm,	Y =  55.000  mm,	Z =   0.600 mm,
	W =180.000 deg,	P =   0.000 deg,	R =    90.000 deg
};
P[3237]{
   GP1:
	UF : 1, UT : 1,		CONFIG : 'N U T, 0, 0, 1',
	X =  100.000  mm,	Y =  55.000  mm,	Z =   15.000 mm,
	W =180.000 deg,	P =   0.000 deg,	R =    90.000 deg
};
P[3238]{
   GP1:
	UF : 1, UT : 1,		CONFIG : 'N U T, 0, 0, 1',
	X =  103.000  mm,	Y =  55.000  mm,	Z =   15.000 mm,
	W =180.000 deg,	P =   0.000 deg,	R =    90.000 deg
};
P[3239]{
   GP1:
	UF : 1, UT : 1,		CONFIG : 'N U T, 0, 0, 1',
	X =  103.000  mm,	Y =  55.000  mm,	Z =   0.600 mm,
	W =180.000 deg,	P =   0.000 deg,	R =    90.000 deg
};
P[3240]{
   GP1:
	UF : 1, UT : 1,		CONFIG : 'N U T, 0, 0, 1',
	X =  103.000  mm,	Y =  55.000  mm,	Z =   15.000 mm,
	W =180.000 deg,	P =   0.000 deg,	R =    90.000 deg
};
P[3241]{
   GP1:
	UF : 1, UT : 1,		CONFIG : 'N U T, 0, 0, 1',
	X =  106.000  mm,	Y =  55.000  mm,	Z =   15.000 mm,
	W =180.000 deg,	P =   0.000 deg,	R =    90.000 deg
};
P[3242]{
   GP1:
	UF : 1, UT : 1,		CONFIG : 'N U T, 0, 0, 1',
	X =  106.000  mm,	Y =  55.000  mm,	Z =   0.600 mm,
	W =180.000 deg,	P =   0.000 deg,	R =    90.000 deg
};
P[3243]{
   GP1:
	UF : 1, UT : 1,		CONFIG : 'N U T, 0, 0, 1',
	X =  106.000  mm,	Y =  55.000  mm,	Z =   15.000 mm,
	W =180.000 deg,	P =   0.000 deg,	R =    90.000 deg
};
P[3244]{
   GP1:
	UF : 1, UT : 1,		CONFIG : 'N U T, 0, 0, 1',
	X =  109.000  mm,	Y =  55.000  mm,	Z =   15.000 mm,
	W =180.000 deg,	P =   0.000 deg,	R =    90.000 deg
};
P[3245]{
   GP1:
	UF : 1, UT : 1,		CONFIG : 'N U T, 0, 0, 1',
	X =  109.000  mm,	Y =  55.000  mm,	Z =   0.600 mm,
	W =180.000 deg,	P =   0.000 deg,	R =    90.000 deg
};
P[3246]{
   GP1:
	UF : 1, UT : 1,		CONFIG : 'N U T, 0, 0, 1',
	X =  109.000  mm,	Y =  55.000  mm,	Z =   15.000 mm,
	W =180.000 deg,	P =   0.000 deg,	R =    90.000 deg
};
P[3247]{
   GP1:
	UF : 1, UT : 1,		CONFIG : 'N U T, 0, 0, 1',
	X =  112.000  mm,	Y =  55.000  mm,	Z =   15.000 mm,
	W =180.000 deg,	P =   0.000 deg,	R =    90.000 deg
};
P[3248]{
   GP1:
	UF : 1, UT : 1,		CONFIG : 'N U T, 0, 0, 1',
	X =  112.000  mm,	Y =  55.000  mm,	Z =   0.600 mm,
	W =180.000 deg,	P =   0.000 deg,	R =    90.000 deg
};
P[3249]{
   GP1:
	UF : 1, UT : 1,		CONFIG : 'N U T, 0, 0, 1',
	X =  112.000  mm,	Y =  55.000  mm,	Z =   15.000 mm,
	W =180.000 deg,	P =   0.000 deg,	R =    90.000 deg
};
P[3259]{
   GP1:
	UF : 1, UT : 1,		CONFIG : 'N U T, 0, 0, 1',
	X =  130.000  mm,	Y =  55.000  mm,	Z =   15.000 mm,
	W =180.000 deg,	P =   0.000 deg,	R =    90.000 deg
};
P[3260]{
   GP1:
	UF : 1, UT : 1,		CONFIG : 'N U T, 0, 0, 1',
	X =  130.000  mm,	Y =  55.000  mm,	Z =   0.600 mm,
	W =180.000 deg,	P =   0.000 deg,	R =    90.000 deg
};
P[3261]{
   GP1:
	UF : 1, UT : 1,		CONFIG : 'N U T, 0, 0, 1',
	X =  130.000  mm,	Y =  55.000  mm,	Z =   15.000 mm,
	W =180.000 deg,	P =   0.000 deg,	R =    90.000 deg
};
P[3262]{
   GP1:
	UF : 1, UT : 1,		CONFIG : 'N U T, 0, 0, 1',
	X =  139.000  mm,	Y =  55.000  mm,	Z =   15.000 mm,
	W =180.000 deg,	P =   0.000 deg,	R =    90.000 deg
};
P[3263]{
   GP1:
	UF : 1, UT : 1,		CONFIG : 'N U T, 0, 0, 1',
	X =  139.000  mm,	Y =  55.000  mm,	Z =   0.600 mm,
	W =180.000 deg,	P =   0.000 deg,	R =    90.000 deg
};
P[3264]{
   GP1:
	UF : 1, UT : 1,		CONFIG : 'N U T, 0, 0, 1',
	X =  139.000  mm,	Y =  55.000  mm,	Z =   15.000 mm,
	W =180.000 deg,	P =   0.000 deg,	R =    90.000 deg
};
P[3268]{
   GP1:
	UF : 1, UT : 1,		CONFIG : 'N U T, 0, 0, 1',
	X =  145.000  mm,	Y =  55.000  mm,	Z =   15.000 mm,
	W =180.000 deg,	P =   0.000 deg,	R =    90.000 deg
};
P[3269]{
   GP1:
	UF : 1, UT : 1,		CONFIG : 'N U T, 0, 0, 1',
	X =  145.000  mm,	Y =  55.000  mm,	Z =   0.600 mm,
	W =180.000 deg,	P =   0.000 deg,	R =    90.000 deg
};
P[3270]{
   GP1:
	UF : 1, UT : 1,		CONFIG : 'N U T, 0, 0, 1',
	X =  145.000  mm,	Y =  55.000  mm,	Z =   15.000 mm,
	W =180.000 deg,	P =   0.000 deg,	R =    90.000 deg
};
P[3277]{
   GP1:
	UF : 1, UT : 1,		CONFIG : 'N U T, 0, 0, 1',
	X =  175.000  mm,	Y =  55.000  mm,	Z =   15.000 mm,
	W =180.000 deg,	P =   0.000 deg,	R =    90.000 deg
};
P[3278]{
   GP1:
	UF : 1, UT : 1,		CONFIG : 'N U T, 0, 0, 1',
	X =  175.000  mm,	Y =  55.000  mm,	Z =   0.600 mm,
	W =180.000 deg,	P =   0.000 deg,	R =    90.000 deg
};
P[3279]{
   GP1:
	UF : 1, UT : 1,		CONFIG : 'N U T, 0, 0, 1',
	X =  175.000  mm,	Y =  55.000  mm,	Z =   15.000 mm,
	W =180.000 deg,	P =   0.000 deg,	R =    90.000 deg
};
P[3280]{
   GP1:
	UF : 1, UT : 1,		CONFIG : 'N U T, 0, 0, 1',
	X =  178.000  mm,	Y =  55.000  mm,	Z =   15.000 mm,
	W =180.000 deg,	P =   0.000 deg,	R =    90.000 deg
};
P[3281]{
   GP1:
	UF : 1, UT : 1,		CONFIG : 'N U T, 0, 0, 1',
	X =  178.000  mm,	Y =  55.000  mm,	Z =   0.600 mm,
	W =180.000 deg,	P =   0.000 deg,	R =    90.000 deg
};
P[3282]{
   GP1:
	UF : 1, UT : 1,		CONFIG : 'N U T, 0, 0, 1',
	X =  178.000  mm,	Y =  55.000  mm,	Z =   15.000 mm,
	W =180.000 deg,	P =   0.000 deg,	R =    90.000 deg
};
P[3283]{
   GP1:
	UF : 1, UT : 1,		CONFIG : 'N U T, 0, 0, 1',
	X =  1.000  mm,	Y =  58.000  mm,	Z =   15.000 mm,
	W =180.000 deg,	P =   0.000 deg,	R =    90.000 deg
};
P[3284]{
   GP1:
	UF : 1, UT : 1,		CONFIG : 'N U T, 0, 0, 1',
	X =  1.000  mm,	Y =  58.000  mm,	Z =   0.600 mm,
	W =180.000 deg,	P =   0.000 deg,	R =    90.000 deg
};
P[3285]{
   GP1:
	UF : 1, UT : 1,		CONFIG : 'N U T, 0, 0, 1',
	X =  1.000  mm,	Y =  58.000  mm,	Z =   15.000 mm,
	W =180.000 deg,	P =   0.000 deg,	R =    90.000 deg
};
P[3286]{
   GP1:
	UF : 1, UT : 1,		CONFIG : 'N U T, 0, 0, 1',
	X =  4.000  mm,	Y =  58.000  mm,	Z =   15.000 mm,
	W =180.000 deg,	P =   0.000 deg,	R =    90.000 deg
};
P[3287]{
   GP1:
	UF : 1, UT : 1,		CONFIG : 'N U T, 0, 0, 1',
	X =  4.000  mm,	Y =  58.000  mm,	Z =   0.600 mm,
	W =180.000 deg,	P =   0.000 deg,	R =    90.000 deg
};
P[3288]{
   GP1:
	UF : 1, UT : 1,		CONFIG : 'N U T, 0, 0, 1',
	X =  4.000  mm,	Y =  58.000  mm,	Z =   15.000 mm,
	W =180.000 deg,	P =   0.000 deg,	R =    90.000 deg
};
P[3289]{
   GP1:
	UF : 1, UT : 1,		CONFIG : 'N U T, 0, 0, 1',
	X =  7.000  mm,	Y =  58.000  mm,	Z =   15.000 mm,
	W =180.000 deg,	P =   0.000 deg,	R =    90.000 deg
};
P[3290]{
   GP1:
	UF : 1, UT : 1,		CONFIG : 'N U T, 0, 0, 1',
	X =  7.000  mm,	Y =  58.000  mm,	Z =   0.600 mm,
	W =180.000 deg,	P =   0.000 deg,	R =    90.000 deg
};
P[3291]{
   GP1:
	UF : 1, UT : 1,		CONFIG : 'N U T, 0, 0, 1',
	X =  7.000  mm,	Y =  58.000  mm,	Z =   15.000 mm,
	W =180.000 deg,	P =   0.000 deg,	R =    90.000 deg
};
P[3292]{
   GP1:
	UF : 1, UT : 1,		CONFIG : 'N U T, 0, 0, 1',
	X =  10.000  mm,	Y =  58.000  mm,	Z =   15.000 mm,
	W =180.000 deg,	P =   0.000 deg,	R =    90.000 deg
};
P[3293]{
   GP1:
	UF : 1, UT : 1,		CONFIG : 'N U T, 0, 0, 1',
	X =  10.000  mm,	Y =  58.000  mm,	Z =   0.600 mm,
	W =180.000 deg,	P =   0.000 deg,	R =    90.000 deg
};
P[3294]{
   GP1:
	UF : 1, UT : 1,		CONFIG : 'N U T, 0, 0, 1',
	X =  10.000  mm,	Y =  58.000  mm,	Z =   15.000 mm,
	W =180.000 deg,	P =   0.000 deg,	R =    90.000 deg
};
P[3295]{
   GP1:
	UF : 1, UT : 1,		CONFIG : 'N U T, 0, 0, 1',
	X =  13.000  mm,	Y =  58.000  mm,	Z =   15.000 mm,
	W =180.000 deg,	P =   0.000 deg,	R =    90.000 deg
};
P[3296]{
   GP1:
	UF : 1, UT : 1,		CONFIG : 'N U T, 0, 0, 1',
	X =  13.000  mm,	Y =  58.000  mm,	Z =   0.600 mm,
	W =180.000 deg,	P =   0.000 deg,	R =    90.000 deg
};
P[3297]{
   GP1:
	UF : 1, UT : 1,		CONFIG : 'N U T, 0, 0, 1',
	X =  13.000  mm,	Y =  58.000  mm,	Z =   15.000 mm,
	W =180.000 deg,	P =   0.000 deg,	R =    90.000 deg
};
P[3298]{
   GP1:
	UF : 1, UT : 1,		CONFIG : 'N U T, 0, 0, 1',
	X =  16.000  mm,	Y =  58.000  mm,	Z =   15.000 mm,
	W =180.000 deg,	P =   0.000 deg,	R =    90.000 deg
};
P[3299]{
   GP1:
	UF : 1, UT : 1,		CONFIG : 'N U T, 0, 0, 1',
	X =  16.000  mm,	Y =  58.000  mm,	Z =   0.600 mm,
	W =180.000 deg,	P =   0.000 deg,	R =    90.000 deg
};
P[3300]{
   GP1:
	UF : 1, UT : 1,		CONFIG : 'N U T, 0, 0, 1',
	X =  16.000  mm,	Y =  58.000  mm,	Z =   15.000 mm,
	W =180.000 deg,	P =   0.000 deg,	R =    90.000 deg
};
P[3301]{
   GP1:
	UF : 1, UT : 1,		CONFIG : 'N U T, 0, 0, 1',
	X =  19.000  mm,	Y =  58.000  mm,	Z =   15.000 mm,
	W =180.000 deg,	P =   0.000 deg,	R =    90.000 deg
};
P[3302]{
   GP1:
	UF : 1, UT : 1,		CONFIG : 'N U T, 0, 0, 1',
	X =  19.000  mm,	Y =  58.000  mm,	Z =   0.600 mm,
	W =180.000 deg,	P =   0.000 deg,	R =    90.000 deg
};
P[3303]{
   GP1:
	UF : 1, UT : 1,		CONFIG : 'N U T, 0, 0, 1',
	X =  19.000  mm,	Y =  58.000  mm,	Z =   15.000 mm,
	W =180.000 deg,	P =   0.000 deg,	R =    90.000 deg
};
P[3304]{
   GP1:
	UF : 1, UT : 1,		CONFIG : 'N U T, 0, 0, 1',
	X =  22.000  mm,	Y =  58.000  mm,	Z =   15.000 mm,
	W =180.000 deg,	P =   0.000 deg,	R =    90.000 deg
};
P[3305]{
   GP1:
	UF : 1, UT : 1,		CONFIG : 'N U T, 0, 0, 1',
	X =  22.000  mm,	Y =  58.000  mm,	Z =   0.600 mm,
	W =180.000 deg,	P =   0.000 deg,	R =    90.000 deg
};
P[3306]{
   GP1:
	UF : 1, UT : 1,		CONFIG : 'N U T, 0, 0, 1',
	X =  22.000  mm,	Y =  58.000  mm,	Z =   15.000 mm,
	W =180.000 deg,	P =   0.000 deg,	R =    90.000 deg
};
P[3307]{
   GP1:
	UF : 1, UT : 1,		CONFIG : 'N U T, 0, 0, 1',
	X =  28.000  mm,	Y =  58.000  mm,	Z =   15.000 mm,
	W =180.000 deg,	P =   0.000 deg,	R =    90.000 deg
};
P[3308]{
   GP1:
	UF : 1, UT : 1,		CONFIG : 'N U T, 0, 0, 1',
	X =  28.000  mm,	Y =  58.000  mm,	Z =   0.600 mm,
	W =180.000 deg,	P =   0.000 deg,	R =    90.000 deg
};
P[3309]{
   GP1:
	UF : 1, UT : 1,		CONFIG : 'N U T, 0, 0, 1',
	X =  28.000  mm,	Y =  58.000  mm,	Z =   15.000 mm,
	W =180.000 deg,	P =   0.000 deg,	R =    90.000 deg
};
P[3310]{
   GP1:
	UF : 1, UT : 1,		CONFIG : 'N U T, 0, 0, 1',
	X =  31.000  mm,	Y =  58.000  mm,	Z =   15.000 mm,
	W =180.000 deg,	P =   0.000 deg,	R =    90.000 deg
};
P[3311]{
   GP1:
	UF : 1, UT : 1,		CONFIG : 'N U T, 0, 0, 1',
	X =  31.000  mm,	Y =  58.000  mm,	Z =   0.600 mm,
	W =180.000 deg,	P =   0.000 deg,	R =    90.000 deg
};
P[3312]{
   GP1:
	UF : 1, UT : 1,		CONFIG : 'N U T, 0, 0, 1',
	X =  31.000  mm,	Y =  58.000  mm,	Z =   15.000 mm,
	W =180.000 deg,	P =   0.000 deg,	R =    90.000 deg
};
P[3313]{
   GP1:
	UF : 1, UT : 1,		CONFIG : 'N U T, 0, 0, 1',
	X =  34.000  mm,	Y =  58.000  mm,	Z =   15.000 mm,
	W =180.000 deg,	P =   0.000 deg,	R =    90.000 deg
};
P[3314]{
   GP1:
	UF : 1, UT : 1,		CONFIG : 'N U T, 0, 0, 1',
	X =  34.000  mm,	Y =  58.000  mm,	Z =   0.600 mm,
	W =180.000 deg,	P =   0.000 deg,	R =    90.000 deg
};
P[3315]{
   GP1:
	UF : 1, UT : 1,		CONFIG : 'N U T, 0, 0, 1',
	X =  34.000  mm,	Y =  58.000  mm,	Z =   15.000 mm,
	W =180.000 deg,	P =   0.000 deg,	R =    90.000 deg
};
P[3316]{
   GP1:
	UF : 1, UT : 1,		CONFIG : 'N U T, 0, 0, 1',
	X =  37.000  mm,	Y =  58.000  mm,	Z =   15.000 mm,
	W =180.000 deg,	P =   0.000 deg,	R =    90.000 deg
};
P[3317]{
   GP1:
	UF : 1, UT : 1,		CONFIG : 'N U T, 0, 0, 1',
	X =  37.000  mm,	Y =  58.000  mm,	Z =   0.600 mm,
	W =180.000 deg,	P =   0.000 deg,	R =    90.000 deg
};
P[3318]{
   GP1:
	UF : 1, UT : 1,		CONFIG : 'N U T, 0, 0, 1',
	X =  37.000  mm,	Y =  58.000  mm,	Z =   15.000 mm,
	W =180.000 deg,	P =   0.000 deg,	R =    90.000 deg
};
P[3319]{
   GP1:
	UF : 1, UT : 1,		CONFIG : 'N U T, 0, 0, 1',
	X =  40.000  mm,	Y =  58.000  mm,	Z =   15.000 mm,
	W =180.000 deg,	P =   0.000 deg,	R =    90.000 deg
};
P[3320]{
   GP1:
	UF : 1, UT : 1,		CONFIG : 'N U T, 0, 0, 1',
	X =  40.000  mm,	Y =  58.000  mm,	Z =   0.600 mm,
	W =180.000 deg,	P =   0.000 deg,	R =    90.000 deg
};
P[3321]{
   GP1:
	UF : 1, UT : 1,		CONFIG : 'N U T, 0, 0, 1',
	X =  40.000  mm,	Y =  58.000  mm,	Z =   15.000 mm,
	W =180.000 deg,	P =   0.000 deg,	R =    90.000 deg
};
P[3322]{
   GP1:
	UF : 1, UT : 1,		CONFIG : 'N U T, 0, 0, 1',
	X =  43.000  mm,	Y =  58.000  mm,	Z =   15.000 mm,
	W =180.000 deg,	P =   0.000 deg,	R =    90.000 deg
};
P[3323]{
   GP1:
	UF : 1, UT : 1,		CONFIG : 'N U T, 0, 0, 1',
	X =  43.000  mm,	Y =  58.000  mm,	Z =   0.600 mm,
	W =180.000 deg,	P =   0.000 deg,	R =    90.000 deg
};
P[3324]{
   GP1:
	UF : 1, UT : 1,		CONFIG : 'N U T, 0, 0, 1',
	X =  43.000  mm,	Y =  58.000  mm,	Z =   15.000 mm,
	W =180.000 deg,	P =   0.000 deg,	R =    90.000 deg
};
P[3325]{
   GP1:
	UF : 1, UT : 1,		CONFIG : 'N U T, 0, 0, 1',
	X =  46.000  mm,	Y =  58.000  mm,	Z =   15.000 mm,
	W =180.000 deg,	P =   0.000 deg,	R =    90.000 deg
};
P[3326]{
   GP1:
	UF : 1, UT : 1,		CONFIG : 'N U T, 0, 0, 1',
	X =  46.000  mm,	Y =  58.000  mm,	Z =   0.600 mm,
	W =180.000 deg,	P =   0.000 deg,	R =    90.000 deg
};
P[3327]{
   GP1:
	UF : 1, UT : 1,		CONFIG : 'N U T, 0, 0, 1',
	X =  46.000  mm,	Y =  58.000  mm,	Z =   15.000 mm,
	W =180.000 deg,	P =   0.000 deg,	R =    90.000 deg
};
P[3328]{
   GP1:
	UF : 1, UT : 1,		CONFIG : 'N U T, 0, 0, 1',
	X =  49.000  mm,	Y =  58.000  mm,	Z =   15.000 mm,
	W =180.000 deg,	P =   0.000 deg,	R =    90.000 deg
};
P[3329]{
   GP1:
	UF : 1, UT : 1,		CONFIG : 'N U T, 0, 0, 1',
	X =  49.000  mm,	Y =  58.000  mm,	Z =   0.600 mm,
	W =180.000 deg,	P =   0.000 deg,	R =    90.000 deg
};
P[3330]{
   GP1:
	UF : 1, UT : 1,		CONFIG : 'N U T, 0, 0, 1',
	X =  49.000  mm,	Y =  58.000  mm,	Z =   15.000 mm,
	W =180.000 deg,	P =   0.000 deg,	R =    90.000 deg
};
P[3331]{
   GP1:
	UF : 1, UT : 1,		CONFIG : 'N U T, 0, 0, 1',
	X =  52.000  mm,	Y =  58.000  mm,	Z =   15.000 mm,
	W =180.000 deg,	P =   0.000 deg,	R =    90.000 deg
};
P[3332]{
   GP1:
	UF : 1, UT : 1,		CONFIG : 'N U T, 0, 0, 1',
	X =  52.000  mm,	Y =  58.000  mm,	Z =   0.600 mm,
	W =180.000 deg,	P =   0.000 deg,	R =    90.000 deg
};
P[3333]{
   GP1:
	UF : 1, UT : 1,		CONFIG : 'N U T, 0, 0, 1',
	X =  52.000  mm,	Y =  58.000  mm,	Z =   15.000 mm,
	W =180.000 deg,	P =   0.000 deg,	R =    90.000 deg
};
P[3334]{
   GP1:
	UF : 1, UT : 1,		CONFIG : 'N U T, 0, 0, 1',
	X =  55.000  mm,	Y =  58.000  mm,	Z =   15.000 mm,
	W =180.000 deg,	P =   0.000 deg,	R =    90.000 deg
};
P[3335]{
   GP1:
	UF : 1, UT : 1,		CONFIG : 'N U T, 0, 0, 1',
	X =  55.000  mm,	Y =  58.000  mm,	Z =   0.600 mm,
	W =180.000 deg,	P =   0.000 deg,	R =    90.000 deg
};
P[3336]{
   GP1:
	UF : 1, UT : 1,		CONFIG : 'N U T, 0, 0, 1',
	X =  55.000  mm,	Y =  58.000  mm,	Z =   15.000 mm,
	W =180.000 deg,	P =   0.000 deg,	R =    90.000 deg
};
P[3337]{
   GP1:
	UF : 1, UT : 1,		CONFIG : 'N U T, 0, 0, 1',
	X =  58.000  mm,	Y =  58.000  mm,	Z =   15.000 mm,
	W =180.000 deg,	P =   0.000 deg,	R =    90.000 deg
};
P[3338]{
   GP1:
	UF : 1, UT : 1,		CONFIG : 'N U T, 0, 0, 1',
	X =  58.000  mm,	Y =  58.000  mm,	Z =   0.600 mm,
	W =180.000 deg,	P =   0.000 deg,	R =    90.000 deg
};
P[3339]{
   GP1:
	UF : 1, UT : 1,		CONFIG : 'N U T, 0, 0, 1',
	X =  58.000  mm,	Y =  58.000  mm,	Z =   15.000 mm,
	W =180.000 deg,	P =   0.000 deg,	R =    90.000 deg
};
P[3358]{
   GP1:
	UF : 1, UT : 1,		CONFIG : 'N U T, 0, 0, 1',
	X =  79.000  mm,	Y =  58.000  mm,	Z =   15.000 mm,
	W =180.000 deg,	P =   0.000 deg,	R =    90.000 deg
};
P[3359]{
   GP1:
	UF : 1, UT : 1,		CONFIG : 'N U T, 0, 0, 1',
	X =  79.000  mm,	Y =  58.000  mm,	Z =   0.600 mm,
	W =180.000 deg,	P =   0.000 deg,	R =    90.000 deg
};
P[3360]{
   GP1:
	UF : 1, UT : 1,		CONFIG : 'N U T, 0, 0, 1',
	X =  79.000  mm,	Y =  58.000  mm,	Z =   15.000 mm,
	W =180.000 deg,	P =   0.000 deg,	R =    90.000 deg
};
P[3364]{
   GP1:
	UF : 1, UT : 1,		CONFIG : 'N U T, 0, 0, 1',
	X =  85.000  mm,	Y =  58.000  mm,	Z =   15.000 mm,
	W =180.000 deg,	P =   0.000 deg,	R =    90.000 deg
};
P[3365]{
   GP1:
	UF : 1, UT : 1,		CONFIG : 'N U T, 0, 0, 1',
	X =  85.000  mm,	Y =  58.000  mm,	Z =   0.600 mm,
	W =180.000 deg,	P =   0.000 deg,	R =    90.000 deg
};
P[3366]{
   GP1:
	UF : 1, UT : 1,		CONFIG : 'N U T, 0, 0, 1',
	X =  85.000  mm,	Y =  58.000  mm,	Z =   15.000 mm,
	W =180.000 deg,	P =   0.000 deg,	R =    90.000 deg
};
P[3367]{
   GP1:
	UF : 1, UT : 1,		CONFIG : 'N U T, 0, 0, 1',
	X =  88.000  mm,	Y =  58.000  mm,	Z =   15.000 mm,
	W =180.000 deg,	P =   0.000 deg,	R =    90.000 deg
};
P[3368]{
   GP1:
	UF : 1, UT : 1,		CONFIG : 'N U T, 0, 0, 1',
	X =  88.000  mm,	Y =  58.000  mm,	Z =   0.600 mm,
	W =180.000 deg,	P =   0.000 deg,	R =    90.000 deg
};
P[3369]{
   GP1:
	UF : 1, UT : 1,		CONFIG : 'N U T, 0, 0, 1',
	X =  88.000  mm,	Y =  58.000  mm,	Z =   15.000 mm,
	W =180.000 deg,	P =   0.000 deg,	R =    90.000 deg
};
P[3370]{
   GP1:
	UF : 1, UT : 1,		CONFIG : 'N U T, 0, 0, 1',
	X =  91.000  mm,	Y =  58.000  mm,	Z =   15.000 mm,
	W =180.000 deg,	P =   0.000 deg,	R =    90.000 deg
};
P[3371]{
   GP1:
	UF : 1, UT : 1,		CONFIG : 'N U T, 0, 0, 1',
	X =  91.000  mm,	Y =  58.000  mm,	Z =   0.600 mm,
	W =180.000 deg,	P =   0.000 deg,	R =    90.000 deg
};
P[3372]{
   GP1:
	UF : 1, UT : 1,		CONFIG : 'N U T, 0, 0, 1',
	X =  91.000  mm,	Y =  58.000  mm,	Z =   15.000 mm,
	W =180.000 deg,	P =   0.000 deg,	R =    90.000 deg
};
P[3373]{
   GP1:
	UF : 1, UT : 1,		CONFIG : 'N U T, 0, 0, 1',
	X =  94.000  mm,	Y =  58.000  mm,	Z =   15.000 mm,
	W =180.000 deg,	P =   0.000 deg,	R =    90.000 deg
};
P[3374]{
   GP1:
	UF : 1, UT : 1,		CONFIG : 'N U T, 0, 0, 1',
	X =  94.000  mm,	Y =  58.000  mm,	Z =   0.600 mm,
	W =180.000 deg,	P =   0.000 deg,	R =    90.000 deg
};
P[3375]{
   GP1:
	UF : 1, UT : 1,		CONFIG : 'N U T, 0, 0, 1',
	X =  94.000  mm,	Y =  58.000  mm,	Z =   15.000 mm,
	W =180.000 deg,	P =   0.000 deg,	R =    90.000 deg
};
P[3376]{
   GP1:
	UF : 1, UT : 1,		CONFIG : 'N U T, 0, 0, 1',
	X =  97.000  mm,	Y =  58.000  mm,	Z =   15.000 mm,
	W =180.000 deg,	P =   0.000 deg,	R =    90.000 deg
};
P[3377]{
   GP1:
	UF : 1, UT : 1,		CONFIG : 'N U T, 0, 0, 1',
	X =  97.000  mm,	Y =  58.000  mm,	Z =   0.600 mm,
	W =180.000 deg,	P =   0.000 deg,	R =    90.000 deg
};
P[3378]{
   GP1:
	UF : 1, UT : 1,		CONFIG : 'N U T, 0, 0, 1',
	X =  97.000  mm,	Y =  58.000  mm,	Z =   15.000 mm,
	W =180.000 deg,	P =   0.000 deg,	R =    90.000 deg
};
P[3379]{
   GP1:
	UF : 1, UT : 1,		CONFIG : 'N U T, 0, 0, 1',
	X =  100.000  mm,	Y =  58.000  mm,	Z =   15.000 mm,
	W =180.000 deg,	P =   0.000 deg,	R =    90.000 deg
};
P[3380]{
   GP1:
	UF : 1, UT : 1,		CONFIG : 'N U T, 0, 0, 1',
	X =  100.000  mm,	Y =  58.000  mm,	Z =   0.600 mm,
	W =180.000 deg,	P =   0.000 deg,	R =    90.000 deg
};
P[3381]{
   GP1:
	UF : 1, UT : 1,		CONFIG : 'N U T, 0, 0, 1',
	X =  100.000  mm,	Y =  58.000  mm,	Z =   15.000 mm,
	W =180.000 deg,	P =   0.000 deg,	R =    90.000 deg
};
P[3382]{
   GP1:
	UF : 1, UT : 1,		CONFIG : 'N U T, 0, 0, 1',
	X =  103.000  mm,	Y =  58.000  mm,	Z =   15.000 mm,
	W =180.000 deg,	P =   0.000 deg,	R =    90.000 deg
};
P[3383]{
   GP1:
	UF : 1, UT : 1,		CONFIG : 'N U T, 0, 0, 1',
	X =  103.000  mm,	Y =  58.000  mm,	Z =   0.600 mm,
	W =180.000 deg,	P =   0.000 deg,	R =    90.000 deg
};
P[3384]{
   GP1:
	UF : 1, UT : 1,		CONFIG : 'N U T, 0, 0, 1',
	X =  103.000  mm,	Y =  58.000  mm,	Z =   15.000 mm,
	W =180.000 deg,	P =   0.000 deg,	R =    90.000 deg
};
P[3385]{
   GP1:
	UF : 1, UT : 1,		CONFIG : 'N U T, 0, 0, 1',
	X =  106.000  mm,	Y =  58.000  mm,	Z =   15.000 mm,
	W =180.000 deg,	P =   0.000 deg,	R =    90.000 deg
};
P[3386]{
   GP1:
	UF : 1, UT : 1,		CONFIG : 'N U T, 0, 0, 1',
	X =  106.000  mm,	Y =  58.000  mm,	Z =   0.600 mm,
	W =180.000 deg,	P =   0.000 deg,	R =    90.000 deg
};
P[3387]{
   GP1:
	UF : 1, UT : 1,		CONFIG : 'N U T, 0, 0, 1',
	X =  106.000  mm,	Y =  58.000  mm,	Z =   15.000 mm,
	W =180.000 deg,	P =   0.000 deg,	R =    90.000 deg
};
P[3388]{
   GP1:
	UF : 1, UT : 1,		CONFIG : 'N U T, 0, 0, 1',
	X =  109.000  mm,	Y =  58.000  mm,	Z =   15.000 mm,
	W =180.000 deg,	P =   0.000 deg,	R =    90.000 deg
};
P[3389]{
   GP1:
	UF : 1, UT : 1,		CONFIG : 'N U T, 0, 0, 1',
	X =  109.000  mm,	Y =  58.000  mm,	Z =   0.600 mm,
	W =180.000 deg,	P =   0.000 deg,	R =    90.000 deg
};
P[3390]{
   GP1:
	UF : 1, UT : 1,		CONFIG : 'N U T, 0, 0, 1',
	X =  109.000  mm,	Y =  58.000  mm,	Z =   15.000 mm,
	W =180.000 deg,	P =   0.000 deg,	R =    90.000 deg
};
P[3391]{
   GP1:
	UF : 1, UT : 1,		CONFIG : 'N U T, 0, 0, 1',
	X =  112.000  mm,	Y =  58.000  mm,	Z =   15.000 mm,
	W =180.000 deg,	P =   0.000 deg,	R =    90.000 deg
};
P[3392]{
   GP1:
	UF : 1, UT : 1,		CONFIG : 'N U T, 0, 0, 1',
	X =  112.000  mm,	Y =  58.000  mm,	Z =   0.600 mm,
	W =180.000 deg,	P =   0.000 deg,	R =    90.000 deg
};
P[3393]{
   GP1:
	UF : 1, UT : 1,		CONFIG : 'N U T, 0, 0, 1',
	X =  112.000  mm,	Y =  58.000  mm,	Z =   15.000 mm,
	W =180.000 deg,	P =   0.000 deg,	R =    90.000 deg
};
P[3400]{
   GP1:
	UF : 1, UT : 1,		CONFIG : 'N U T, 0, 0, 1',
	X =  127.000  mm,	Y =  58.000  mm,	Z =   15.000 mm,
	W =180.000 deg,	P =   0.000 deg,	R =    90.000 deg
};
P[3401]{
   GP1:
	UF : 1, UT : 1,		CONFIG : 'N U T, 0, 0, 1',
	X =  127.000  mm,	Y =  58.000  mm,	Z =   0.600 mm,
	W =180.000 deg,	P =   0.000 deg,	R =    90.000 deg
};
P[3402]{
   GP1:
	UF : 1, UT : 1,		CONFIG : 'N U T, 0, 0, 1',
	X =  127.000  mm,	Y =  58.000  mm,	Z =   15.000 mm,
	W =180.000 deg,	P =   0.000 deg,	R =    90.000 deg
};
P[3406]{
   GP1:
	UF : 1, UT : 1,		CONFIG : 'N U T, 0, 0, 1',
	X =  136.000  mm,	Y =  58.000  mm,	Z =   15.000 mm,
	W =180.000 deg,	P =   0.000 deg,	R =    90.000 deg
};
P[3407]{
   GP1:
	UF : 1, UT : 1,		CONFIG : 'N U T, 0, 0, 1',
	X =  136.000  mm,	Y =  58.000  mm,	Z =   0.600 mm,
	W =180.000 deg,	P =   0.000 deg,	R =    90.000 deg
};
P[3408]{
   GP1:
	UF : 1, UT : 1,		CONFIG : 'N U T, 0, 0, 1',
	X =  136.000  mm,	Y =  58.000  mm,	Z =   15.000 mm,
	W =180.000 deg,	P =   0.000 deg,	R =    90.000 deg
};
P[3409]{
   GP1:
	UF : 1, UT : 1,		CONFIG : 'N U T, 0, 0, 1',
	X =  142.000  mm,	Y =  58.000  mm,	Z =   15.000 mm,
	W =180.000 deg,	P =   0.000 deg,	R =    90.000 deg
};
P[3410]{
   GP1:
	UF : 1, UT : 1,		CONFIG : 'N U T, 0, 0, 1',
	X =  142.000  mm,	Y =  58.000  mm,	Z =   0.600 mm,
	W =180.000 deg,	P =   0.000 deg,	R =    90.000 deg
};
P[3411]{
   GP1:
	UF : 1, UT : 1,		CONFIG : 'N U T, 0, 0, 1',
	X =  142.000  mm,	Y =  58.000  mm,	Z =   15.000 mm,
	W =180.000 deg,	P =   0.000 deg,	R =    90.000 deg
};
P[3421]{
   GP1:
	UF : 1, UT : 1,		CONFIG : 'N U T, 0, 0, 1',
	X =  175.000  mm,	Y =  58.000  mm,	Z =   15.000 mm,
	W =180.000 deg,	P =   0.000 deg,	R =    90.000 deg
};
P[3422]{
   GP1:
	UF : 1, UT : 1,		CONFIG : 'N U T, 0, 0, 1',
	X =  175.000  mm,	Y =  58.000  mm,	Z =   0.600 mm,
	W =180.000 deg,	P =   0.000 deg,	R =    90.000 deg
};
P[3423]{
   GP1:
	UF : 1, UT : 1,		CONFIG : 'N U T, 0, 0, 1',
	X =  175.000  mm,	Y =  58.000  mm,	Z =   15.000 mm,
	W =180.000 deg,	P =   0.000 deg,	R =    90.000 deg
};
P[3424]{
   GP1:
	UF : 1, UT : 1,		CONFIG : 'N U T, 0, 0, 1',
	X =  178.000  mm,	Y =  58.000  mm,	Z =   15.000 mm,
	W =180.000 deg,	P =   0.000 deg,	R =    90.000 deg
};
P[3425]{
   GP1:
	UF : 1, UT : 1,		CONFIG : 'N U T, 0, 0, 1',
	X =  178.000  mm,	Y =  58.000  mm,	Z =   0.600 mm,
	W =180.000 deg,	P =   0.000 deg,	R =    90.000 deg
};
P[3426]{
   GP1:
	UF : 1, UT : 1,		CONFIG : 'N U T, 0, 0, 1',
	X =  178.000  mm,	Y =  58.000  mm,	Z =   15.000 mm,
	W =180.000 deg,	P =   0.000 deg,	R =    90.000 deg
};
P[3427]{
   GP1:
	UF : 1, UT : 1,		CONFIG : 'N U T, 0, 0, 1',
	X =  1.000  mm,	Y =  61.000  mm,	Z =   15.000 mm,
	W =180.000 deg,	P =   0.000 deg,	R =    90.000 deg
};
P[3428]{
   GP1:
	UF : 1, UT : 1,		CONFIG : 'N U T, 0, 0, 1',
	X =  1.000  mm,	Y =  61.000  mm,	Z =   0.600 mm,
	W =180.000 deg,	P =   0.000 deg,	R =    90.000 deg
};
P[3429]{
   GP1:
	UF : 1, UT : 1,		CONFIG : 'N U T, 0, 0, 1',
	X =  1.000  mm,	Y =  61.000  mm,	Z =   15.000 mm,
	W =180.000 deg,	P =   0.000 deg,	R =    90.000 deg
};
P[3430]{
   GP1:
	UF : 1, UT : 1,		CONFIG : 'N U T, 0, 0, 1',
	X =  4.000  mm,	Y =  61.000  mm,	Z =   15.000 mm,
	W =180.000 deg,	P =   0.000 deg,	R =    90.000 deg
};
P[3431]{
   GP1:
	UF : 1, UT : 1,		CONFIG : 'N U T, 0, 0, 1',
	X =  4.000  mm,	Y =  61.000  mm,	Z =   0.600 mm,
	W =180.000 deg,	P =   0.000 deg,	R =    90.000 deg
};
P[3432]{
   GP1:
	UF : 1, UT : 1,		CONFIG : 'N U T, 0, 0, 1',
	X =  4.000  mm,	Y =  61.000  mm,	Z =   15.000 mm,
	W =180.000 deg,	P =   0.000 deg,	R =    90.000 deg
};
P[3433]{
   GP1:
	UF : 1, UT : 1,		CONFIG : 'N U T, 0, 0, 1',
	X =  7.000  mm,	Y =  61.000  mm,	Z =   15.000 mm,
	W =180.000 deg,	P =   0.000 deg,	R =    90.000 deg
};
P[3434]{
   GP1:
	UF : 1, UT : 1,		CONFIG : 'N U T, 0, 0, 1',
	X =  7.000  mm,	Y =  61.000  mm,	Z =   0.600 mm,
	W =180.000 deg,	P =   0.000 deg,	R =    90.000 deg
};
P[3435]{
   GP1:
	UF : 1, UT : 1,		CONFIG : 'N U T, 0, 0, 1',
	X =  7.000  mm,	Y =  61.000  mm,	Z =   15.000 mm,
	W =180.000 deg,	P =   0.000 deg,	R =    90.000 deg
};
P[3436]{
   GP1:
	UF : 1, UT : 1,		CONFIG : 'N U T, 0, 0, 1',
	X =  10.000  mm,	Y =  61.000  mm,	Z =   15.000 mm,
	W =180.000 deg,	P =   0.000 deg,	R =    90.000 deg
};
P[3437]{
   GP1:
	UF : 1, UT : 1,		CONFIG : 'N U T, 0, 0, 1',
	X =  10.000  mm,	Y =  61.000  mm,	Z =   0.600 mm,
	W =180.000 deg,	P =   0.000 deg,	R =    90.000 deg
};
P[3438]{
   GP1:
	UF : 1, UT : 1,		CONFIG : 'N U T, 0, 0, 1',
	X =  10.000  mm,	Y =  61.000  mm,	Z =   15.000 mm,
	W =180.000 deg,	P =   0.000 deg,	R =    90.000 deg
};
P[3439]{
   GP1:
	UF : 1, UT : 1,		CONFIG : 'N U T, 0, 0, 1',
	X =  13.000  mm,	Y =  61.000  mm,	Z =   15.000 mm,
	W =180.000 deg,	P =   0.000 deg,	R =    90.000 deg
};
P[3440]{
   GP1:
	UF : 1, UT : 1,		CONFIG : 'N U T, 0, 0, 1',
	X =  13.000  mm,	Y =  61.000  mm,	Z =   0.600 mm,
	W =180.000 deg,	P =   0.000 deg,	R =    90.000 deg
};
P[3441]{
   GP1:
	UF : 1, UT : 1,		CONFIG : 'N U T, 0, 0, 1',
	X =  13.000  mm,	Y =  61.000  mm,	Z =   15.000 mm,
	W =180.000 deg,	P =   0.000 deg,	R =    90.000 deg
};
P[3442]{
   GP1:
	UF : 1, UT : 1,		CONFIG : 'N U T, 0, 0, 1',
	X =  16.000  mm,	Y =  61.000  mm,	Z =   15.000 mm,
	W =180.000 deg,	P =   0.000 deg,	R =    90.000 deg
};
P[3443]{
   GP1:
	UF : 1, UT : 1,		CONFIG : 'N U T, 0, 0, 1',
	X =  16.000  mm,	Y =  61.000  mm,	Z =   0.600 mm,
	W =180.000 deg,	P =   0.000 deg,	R =    90.000 deg
};
P[3444]{
   GP1:
	UF : 1, UT : 1,		CONFIG : 'N U T, 0, 0, 1',
	X =  16.000  mm,	Y =  61.000  mm,	Z =   15.000 mm,
	W =180.000 deg,	P =   0.000 deg,	R =    90.000 deg
};
P[3445]{
   GP1:
	UF : 1, UT : 1,		CONFIG : 'N U T, 0, 0, 1',
	X =  19.000  mm,	Y =  61.000  mm,	Z =   15.000 mm,
	W =180.000 deg,	P =   0.000 deg,	R =    90.000 deg
};
P[3446]{
   GP1:
	UF : 1, UT : 1,		CONFIG : 'N U T, 0, 0, 1',
	X =  19.000  mm,	Y =  61.000  mm,	Z =   0.600 mm,
	W =180.000 deg,	P =   0.000 deg,	R =    90.000 deg
};
P[3447]{
   GP1:
	UF : 1, UT : 1,		CONFIG : 'N U T, 0, 0, 1',
	X =  19.000  mm,	Y =  61.000  mm,	Z =   15.000 mm,
	W =180.000 deg,	P =   0.000 deg,	R =    90.000 deg
};
P[3448]{
   GP1:
	UF : 1, UT : 1,		CONFIG : 'N U T, 0, 0, 1',
	X =  22.000  mm,	Y =  61.000  mm,	Z =   15.000 mm,
	W =180.000 deg,	P =   0.000 deg,	R =    90.000 deg
};
P[3449]{
   GP1:
	UF : 1, UT : 1,		CONFIG : 'N U T, 0, 0, 1',
	X =  22.000  mm,	Y =  61.000  mm,	Z =   0.600 mm,
	W =180.000 deg,	P =   0.000 deg,	R =    90.000 deg
};
P[3450]{
   GP1:
	UF : 1, UT : 1,		CONFIG : 'N U T, 0, 0, 1',
	X =  22.000  mm,	Y =  61.000  mm,	Z =   15.000 mm,
	W =180.000 deg,	P =   0.000 deg,	R =    90.000 deg
};
P[3451]{
   GP1:
	UF : 1, UT : 1,		CONFIG : 'N U T, 0, 0, 1',
	X =  28.000  mm,	Y =  61.000  mm,	Z =   15.000 mm,
	W =180.000 deg,	P =   0.000 deg,	R =    90.000 deg
};
P[3452]{
   GP1:
	UF : 1, UT : 1,		CONFIG : 'N U T, 0, 0, 1',
	X =  28.000  mm,	Y =  61.000  mm,	Z =   0.600 mm,
	W =180.000 deg,	P =   0.000 deg,	R =    90.000 deg
};
P[3453]{
   GP1:
	UF : 1, UT : 1,		CONFIG : 'N U T, 0, 0, 1',
	X =  28.000  mm,	Y =  61.000  mm,	Z =   15.000 mm,
	W =180.000 deg,	P =   0.000 deg,	R =    90.000 deg
};
P[3454]{
   GP1:
	UF : 1, UT : 1,		CONFIG : 'N U T, 0, 0, 1',
	X =  31.000  mm,	Y =  61.000  mm,	Z =   15.000 mm,
	W =180.000 deg,	P =   0.000 deg,	R =    90.000 deg
};
P[3455]{
   GP1:
	UF : 1, UT : 1,		CONFIG : 'N U T, 0, 0, 1',
	X =  31.000  mm,	Y =  61.000  mm,	Z =   0.600 mm,
	W =180.000 deg,	P =   0.000 deg,	R =    90.000 deg
};
P[3456]{
   GP1:
	UF : 1, UT : 1,		CONFIG : 'N U T, 0, 0, 1',
	X =  31.000  mm,	Y =  61.000  mm,	Z =   15.000 mm,
	W =180.000 deg,	P =   0.000 deg,	R =    90.000 deg
};
P[3457]{
   GP1:
	UF : 1, UT : 1,		CONFIG : 'N U T, 0, 0, 1',
	X =  34.000  mm,	Y =  61.000  mm,	Z =   15.000 mm,
	W =180.000 deg,	P =   0.000 deg,	R =    90.000 deg
};
P[3458]{
   GP1:
	UF : 1, UT : 1,		CONFIG : 'N U T, 0, 0, 1',
	X =  34.000  mm,	Y =  61.000  mm,	Z =   0.600 mm,
	W =180.000 deg,	P =   0.000 deg,	R =    90.000 deg
};
P[3459]{
   GP1:
	UF : 1, UT : 1,		CONFIG : 'N U T, 0, 0, 1',
	X =  34.000  mm,	Y =  61.000  mm,	Z =   15.000 mm,
	W =180.000 deg,	P =   0.000 deg,	R =    90.000 deg
};
P[3460]{
   GP1:
	UF : 1, UT : 1,		CONFIG : 'N U T, 0, 0, 1',
	X =  37.000  mm,	Y =  61.000  mm,	Z =   15.000 mm,
	W =180.000 deg,	P =   0.000 deg,	R =    90.000 deg
};
P[3461]{
   GP1:
	UF : 1, UT : 1,		CONFIG : 'N U T, 0, 0, 1',
	X =  37.000  mm,	Y =  61.000  mm,	Z =   0.600 mm,
	W =180.000 deg,	P =   0.000 deg,	R =    90.000 deg
};
P[3462]{
   GP1:
	UF : 1, UT : 1,		CONFIG : 'N U T, 0, 0, 1',
	X =  37.000  mm,	Y =  61.000  mm,	Z =   15.000 mm,
	W =180.000 deg,	P =   0.000 deg,	R =    90.000 deg
};
P[3463]{
   GP1:
	UF : 1, UT : 1,		CONFIG : 'N U T, 0, 0, 1',
	X =  40.000  mm,	Y =  61.000  mm,	Z =   15.000 mm,
	W =180.000 deg,	P =   0.000 deg,	R =    90.000 deg
};
P[3464]{
   GP1:
	UF : 1, UT : 1,		CONFIG : 'N U T, 0, 0, 1',
	X =  40.000  mm,	Y =  61.000  mm,	Z =   0.600 mm,
	W =180.000 deg,	P =   0.000 deg,	R =    90.000 deg
};
P[3465]{
   GP1:
	UF : 1, UT : 1,		CONFIG : 'N U T, 0, 0, 1',
	X =  40.000  mm,	Y =  61.000  mm,	Z =   15.000 mm,
	W =180.000 deg,	P =   0.000 deg,	R =    90.000 deg
};
P[3466]{
   GP1:
	UF : 1, UT : 1,		CONFIG : 'N U T, 0, 0, 1',
	X =  43.000  mm,	Y =  61.000  mm,	Z =   15.000 mm,
	W =180.000 deg,	P =   0.000 deg,	R =    90.000 deg
};
P[3467]{
   GP1:
	UF : 1, UT : 1,		CONFIG : 'N U T, 0, 0, 1',
	X =  43.000  mm,	Y =  61.000  mm,	Z =   0.600 mm,
	W =180.000 deg,	P =   0.000 deg,	R =    90.000 deg
};
P[3468]{
   GP1:
	UF : 1, UT : 1,		CONFIG : 'N U T, 0, 0, 1',
	X =  43.000  mm,	Y =  61.000  mm,	Z =   15.000 mm,
	W =180.000 deg,	P =   0.000 deg,	R =    90.000 deg
};
P[3469]{
   GP1:
	UF : 1, UT : 1,		CONFIG : 'N U T, 0, 0, 1',
	X =  46.000  mm,	Y =  61.000  mm,	Z =   15.000 mm,
	W =180.000 deg,	P =   0.000 deg,	R =    90.000 deg
};
P[3470]{
   GP1:
	UF : 1, UT : 1,		CONFIG : 'N U T, 0, 0, 1',
	X =  46.000  mm,	Y =  61.000  mm,	Z =   0.600 mm,
	W =180.000 deg,	P =   0.000 deg,	R =    90.000 deg
};
P[3471]{
   GP1:
	UF : 1, UT : 1,		CONFIG : 'N U T, 0, 0, 1',
	X =  46.000  mm,	Y =  61.000  mm,	Z =   15.000 mm,
	W =180.000 deg,	P =   0.000 deg,	R =    90.000 deg
};
P[3472]{
   GP1:
	UF : 1, UT : 1,		CONFIG : 'N U T, 0, 0, 1',
	X =  49.000  mm,	Y =  61.000  mm,	Z =   15.000 mm,
	W =180.000 deg,	P =   0.000 deg,	R =    90.000 deg
};
P[3473]{
   GP1:
	UF : 1, UT : 1,		CONFIG : 'N U T, 0, 0, 1',
	X =  49.000  mm,	Y =  61.000  mm,	Z =   0.600 mm,
	W =180.000 deg,	P =   0.000 deg,	R =    90.000 deg
};
P[3474]{
   GP1:
	UF : 1, UT : 1,		CONFIG : 'N U T, 0, 0, 1',
	X =  49.000  mm,	Y =  61.000  mm,	Z =   15.000 mm,
	W =180.000 deg,	P =   0.000 deg,	R =    90.000 deg
};
P[3475]{
   GP1:
	UF : 1, UT : 1,		CONFIG : 'N U T, 0, 0, 1',
	X =  52.000  mm,	Y =  61.000  mm,	Z =   15.000 mm,
	W =180.000 deg,	P =   0.000 deg,	R =    90.000 deg
};
P[3476]{
   GP1:
	UF : 1, UT : 1,		CONFIG : 'N U T, 0, 0, 1',
	X =  52.000  mm,	Y =  61.000  mm,	Z =   0.600 mm,
	W =180.000 deg,	P =   0.000 deg,	R =    90.000 deg
};
P[3477]{
   GP1:
	UF : 1, UT : 1,		CONFIG : 'N U T, 0, 0, 1',
	X =  52.000  mm,	Y =  61.000  mm,	Z =   15.000 mm,
	W =180.000 deg,	P =   0.000 deg,	R =    90.000 deg
};
P[3478]{
   GP1:
	UF : 1, UT : 1,		CONFIG : 'N U T, 0, 0, 1',
	X =  55.000  mm,	Y =  61.000  mm,	Z =   15.000 mm,
	W =180.000 deg,	P =   0.000 deg,	R =    90.000 deg
};
P[3479]{
   GP1:
	UF : 1, UT : 1,		CONFIG : 'N U T, 0, 0, 1',
	X =  55.000  mm,	Y =  61.000  mm,	Z =   0.600 mm,
	W =180.000 deg,	P =   0.000 deg,	R =    90.000 deg
};
P[3480]{
   GP1:
	UF : 1, UT : 1,		CONFIG : 'N U T, 0, 0, 1',
	X =  55.000  mm,	Y =  61.000  mm,	Z =   15.000 mm,
	W =180.000 deg,	P =   0.000 deg,	R =    90.000 deg
};
P[3484]{
   GP1:
	UF : 1, UT : 1,		CONFIG : 'N U T, 0, 0, 1',
	X =  61.000  mm,	Y =  61.000  mm,	Z =   15.000 mm,
	W =180.000 deg,	P =   0.000 deg,	R =    90.000 deg
};
P[3485]{
   GP1:
	UF : 1, UT : 1,		CONFIG : 'N U T, 0, 0, 1',
	X =  61.000  mm,	Y =  61.000  mm,	Z =   0.600 mm,
	W =180.000 deg,	P =   0.000 deg,	R =    90.000 deg
};
P[3486]{
   GP1:
	UF : 1, UT : 1,		CONFIG : 'N U T, 0, 0, 1',
	X =  61.000  mm,	Y =  61.000  mm,	Z =   15.000 mm,
	W =180.000 deg,	P =   0.000 deg,	R =    90.000 deg
};
P[3508]{
   GP1:
	UF : 1, UT : 1,		CONFIG : 'N U T, 0, 0, 1',
	X =  85.000  mm,	Y =  61.000  mm,	Z =   15.000 mm,
	W =180.000 deg,	P =   0.000 deg,	R =    90.000 deg
};
P[3509]{
   GP1:
	UF : 1, UT : 1,		CONFIG : 'N U T, 0, 0, 1',
	X =  85.000  mm,	Y =  61.000  mm,	Z =   0.600 mm,
	W =180.000 deg,	P =   0.000 deg,	R =    90.000 deg
};
P[3510]{
   GP1:
	UF : 1, UT : 1,		CONFIG : 'N U T, 0, 0, 1',
	X =  85.000  mm,	Y =  61.000  mm,	Z =   15.000 mm,
	W =180.000 deg,	P =   0.000 deg,	R =    90.000 deg
};
P[3511]{
   GP1:
	UF : 1, UT : 1,		CONFIG : 'N U T, 0, 0, 1',
	X =  88.000  mm,	Y =  61.000  mm,	Z =   15.000 mm,
	W =180.000 deg,	P =   0.000 deg,	R =    90.000 deg
};
P[3512]{
   GP1:
	UF : 1, UT : 1,		CONFIG : 'N U T, 0, 0, 1',
	X =  88.000  mm,	Y =  61.000  mm,	Z =   0.600 mm,
	W =180.000 deg,	P =   0.000 deg,	R =    90.000 deg
};
P[3513]{
   GP1:
	UF : 1, UT : 1,		CONFIG : 'N U T, 0, 0, 1',
	X =  88.000  mm,	Y =  61.000  mm,	Z =   15.000 mm,
	W =180.000 deg,	P =   0.000 deg,	R =    90.000 deg
};
P[3514]{
   GP1:
	UF : 1, UT : 1,		CONFIG : 'N U T, 0, 0, 1',
	X =  91.000  mm,	Y =  61.000  mm,	Z =   15.000 mm,
	W =180.000 deg,	P =   0.000 deg,	R =    90.000 deg
};
P[3515]{
   GP1:
	UF : 1, UT : 1,		CONFIG : 'N U T, 0, 0, 1',
	X =  91.000  mm,	Y =  61.000  mm,	Z =   0.600 mm,
	W =180.000 deg,	P =   0.000 deg,	R =    90.000 deg
};
P[3516]{
   GP1:
	UF : 1, UT : 1,		CONFIG : 'N U T, 0, 0, 1',
	X =  91.000  mm,	Y =  61.000  mm,	Z =   15.000 mm,
	W =180.000 deg,	P =   0.000 deg,	R =    90.000 deg
};
P[3517]{
   GP1:
	UF : 1, UT : 1,		CONFIG : 'N U T, 0, 0, 1',
	X =  94.000  mm,	Y =  61.000  mm,	Z =   15.000 mm,
	W =180.000 deg,	P =   0.000 deg,	R =    90.000 deg
};
P[3518]{
   GP1:
	UF : 1, UT : 1,		CONFIG : 'N U T, 0, 0, 1',
	X =  94.000  mm,	Y =  61.000  mm,	Z =   0.600 mm,
	W =180.000 deg,	P =   0.000 deg,	R =    90.000 deg
};
P[3519]{
   GP1:
	UF : 1, UT : 1,		CONFIG : 'N U T, 0, 0, 1',
	X =  94.000  mm,	Y =  61.000  mm,	Z =   15.000 mm,
	W =180.000 deg,	P =   0.000 deg,	R =    90.000 deg
};
P[3520]{
   GP1:
	UF : 1, UT : 1,		CONFIG : 'N U T, 0, 0, 1',
	X =  97.000  mm,	Y =  61.000  mm,	Z =   15.000 mm,
	W =180.000 deg,	P =   0.000 deg,	R =    90.000 deg
};
P[3521]{
   GP1:
	UF : 1, UT : 1,		CONFIG : 'N U T, 0, 0, 1',
	X =  97.000  mm,	Y =  61.000  mm,	Z =   0.600 mm,
	W =180.000 deg,	P =   0.000 deg,	R =    90.000 deg
};
P[3522]{
   GP1:
	UF : 1, UT : 1,		CONFIG : 'N U T, 0, 0, 1',
	X =  97.000  mm,	Y =  61.000  mm,	Z =   15.000 mm,
	W =180.000 deg,	P =   0.000 deg,	R =    90.000 deg
};
P[3523]{
   GP1:
	UF : 1, UT : 1,		CONFIG : 'N U T, 0, 0, 1',
	X =  100.000  mm,	Y =  61.000  mm,	Z =   15.000 mm,
	W =180.000 deg,	P =   0.000 deg,	R =    90.000 deg
};
P[3524]{
   GP1:
	UF : 1, UT : 1,		CONFIG : 'N U T, 0, 0, 1',
	X =  100.000  mm,	Y =  61.000  mm,	Z =   0.600 mm,
	W =180.000 deg,	P =   0.000 deg,	R =    90.000 deg
};
P[3525]{
   GP1:
	UF : 1, UT : 1,		CONFIG : 'N U T, 0, 0, 1',
	X =  100.000  mm,	Y =  61.000  mm,	Z =   15.000 mm,
	W =180.000 deg,	P =   0.000 deg,	R =    90.000 deg
};
P[3526]{
   GP1:
	UF : 1, UT : 1,		CONFIG : 'N U T, 0, 0, 1',
	X =  103.000  mm,	Y =  61.000  mm,	Z =   15.000 mm,
	W =180.000 deg,	P =   0.000 deg,	R =    90.000 deg
};
P[3527]{
   GP1:
	UF : 1, UT : 1,		CONFIG : 'N U T, 0, 0, 1',
	X =  103.000  mm,	Y =  61.000  mm,	Z =   0.600 mm,
	W =180.000 deg,	P =   0.000 deg,	R =    90.000 deg
};
P[3528]{
   GP1:
	UF : 1, UT : 1,		CONFIG : 'N U T, 0, 0, 1',
	X =  103.000  mm,	Y =  61.000  mm,	Z =   15.000 mm,
	W =180.000 deg,	P =   0.000 deg,	R =    90.000 deg
};
P[3529]{
   GP1:
	UF : 1, UT : 1,		CONFIG : 'N U T, 0, 0, 1',
	X =  106.000  mm,	Y =  61.000  mm,	Z =   15.000 mm,
	W =180.000 deg,	P =   0.000 deg,	R =    90.000 deg
};
P[3530]{
   GP1:
	UF : 1, UT : 1,		CONFIG : 'N U T, 0, 0, 1',
	X =  106.000  mm,	Y =  61.000  mm,	Z =   0.600 mm,
	W =180.000 deg,	P =   0.000 deg,	R =    90.000 deg
};
P[3531]{
   GP1:
	UF : 1, UT : 1,		CONFIG : 'N U T, 0, 0, 1',
	X =  106.000  mm,	Y =  61.000  mm,	Z =   15.000 mm,
	W =180.000 deg,	P =   0.000 deg,	R =    90.000 deg
};
P[3532]{
   GP1:
	UF : 1, UT : 1,		CONFIG : 'N U T, 0, 0, 1',
	X =  109.000  mm,	Y =  61.000  mm,	Z =   15.000 mm,
	W =180.000 deg,	P =   0.000 deg,	R =    90.000 deg
};
P[3533]{
   GP1:
	UF : 1, UT : 1,		CONFIG : 'N U T, 0, 0, 1',
	X =  109.000  mm,	Y =  61.000  mm,	Z =   0.600 mm,
	W =180.000 deg,	P =   0.000 deg,	R =    90.000 deg
};
P[3534]{
   GP1:
	UF : 1, UT : 1,		CONFIG : 'N U T, 0, 0, 1',
	X =  109.000  mm,	Y =  61.000  mm,	Z =   15.000 mm,
	W =180.000 deg,	P =   0.000 deg,	R =    90.000 deg
};
P[3535]{
   GP1:
	UF : 1, UT : 1,		CONFIG : 'N U T, 0, 0, 1',
	X =  112.000  mm,	Y =  61.000  mm,	Z =   15.000 mm,
	W =180.000 deg,	P =   0.000 deg,	R =    90.000 deg
};
P[3536]{
   GP1:
	UF : 1, UT : 1,		CONFIG : 'N U T, 0, 0, 1',
	X =  112.000  mm,	Y =  61.000  mm,	Z =   0.600 mm,
	W =180.000 deg,	P =   0.000 deg,	R =    90.000 deg
};
P[3537]{
   GP1:
	UF : 1, UT : 1,		CONFIG : 'N U T, 0, 0, 1',
	X =  112.000  mm,	Y =  61.000  mm,	Z =   15.000 mm,
	W =180.000 deg,	P =   0.000 deg,	R =    90.000 deg
};
P[3538]{
   GP1:
	UF : 1, UT : 1,		CONFIG : 'N U T, 0, 0, 1',
	X =  115.000  mm,	Y =  61.000  mm,	Z =   15.000 mm,
	W =180.000 deg,	P =   0.000 deg,	R =    90.000 deg
};
P[3539]{
   GP1:
	UF : 1, UT : 1,		CONFIG : 'N U T, 0, 0, 1',
	X =  115.000  mm,	Y =  61.000  mm,	Z =   0.600 mm,
	W =180.000 deg,	P =   0.000 deg,	R =    90.000 deg
};
P[3540]{
   GP1:
	UF : 1, UT : 1,		CONFIG : 'N U T, 0, 0, 1',
	X =  115.000  mm,	Y =  61.000  mm,	Z =   15.000 mm,
	W =180.000 deg,	P =   0.000 deg,	R =    90.000 deg
};
P[3550]{
   GP1:
	UF : 1, UT : 1,		CONFIG : 'N U T, 0, 0, 1',
	X =  133.000  mm,	Y =  61.000  mm,	Z =   15.000 mm,
	W =180.000 deg,	P =   0.000 deg,	R =    90.000 deg
};
P[3551]{
   GP1:
	UF : 1, UT : 1,		CONFIG : 'N U T, 0, 0, 1',
	X =  133.000  mm,	Y =  61.000  mm,	Z =   0.600 mm,
	W =180.000 deg,	P =   0.000 deg,	R =    90.000 deg
};
P[3552]{
   GP1:
	UF : 1, UT : 1,		CONFIG : 'N U T, 0, 0, 1',
	X =  133.000  mm,	Y =  61.000  mm,	Z =   15.000 mm,
	W =180.000 deg,	P =   0.000 deg,	R =    90.000 deg
};
P[3553]{
   GP1:
	UF : 1, UT : 1,		CONFIG : 'N U T, 0, 0, 1',
	X =  139.000  mm,	Y =  61.000  mm,	Z =   15.000 mm,
	W =180.000 deg,	P =   0.000 deg,	R =    90.000 deg
};
P[3554]{
   GP1:
	UF : 1, UT : 1,		CONFIG : 'N U T, 0, 0, 1',
	X =  139.000  mm,	Y =  61.000  mm,	Z =   0.600 mm,
	W =180.000 deg,	P =   0.000 deg,	R =    90.000 deg
};
P[3555]{
   GP1:
	UF : 1, UT : 1,		CONFIG : 'N U T, 0, 0, 1',
	X =  139.000  mm,	Y =  61.000  mm,	Z =   15.000 mm,
	W =180.000 deg,	P =   0.000 deg,	R =    90.000 deg
};
P[3559]{
   GP1:
	UF : 1, UT : 1,		CONFIG : 'N U T, 0, 0, 1',
	X =  145.000  mm,	Y =  61.000  mm,	Z =   15.000 mm,
	W =180.000 deg,	P =   0.000 deg,	R =    90.000 deg
};
P[3560]{
   GP1:
	UF : 1, UT : 1,		CONFIG : 'N U T, 0, 0, 1',
	X =  145.000  mm,	Y =  61.000  mm,	Z =   0.600 mm,
	W =180.000 deg,	P =   0.000 deg,	R =    90.000 deg
};
P[3561]{
   GP1:
	UF : 1, UT : 1,		CONFIG : 'N U T, 0, 0, 1',
	X =  145.000  mm,	Y =  61.000  mm,	Z =   15.000 mm,
	W =180.000 deg,	P =   0.000 deg,	R =    90.000 deg
};
P[3565]{
   GP1:
	UF : 1, UT : 1,		CONFIG : 'N U T, 0, 0, 1',
	X =  175.000  mm,	Y =  61.000  mm,	Z =   15.000 mm,
	W =180.000 deg,	P =   0.000 deg,	R =    90.000 deg
};
P[3566]{
   GP1:
	UF : 1, UT : 1,		CONFIG : 'N U T, 0, 0, 1',
	X =  175.000  mm,	Y =  61.000  mm,	Z =   0.600 mm,
	W =180.000 deg,	P =   0.000 deg,	R =    90.000 deg
};
P[3567]{
   GP1:
	UF : 1, UT : 1,		CONFIG : 'N U T, 0, 0, 1',
	X =  175.000  mm,	Y =  61.000  mm,	Z =   15.000 mm,
	W =180.000 deg,	P =   0.000 deg,	R =    90.000 deg
};
P[3568]{
   GP1:
	UF : 1, UT : 1,		CONFIG : 'N U T, 0, 0, 1',
	X =  178.000  mm,	Y =  61.000  mm,	Z =   15.000 mm,
	W =180.000 deg,	P =   0.000 deg,	R =    90.000 deg
};
P[3569]{
   GP1:
	UF : 1, UT : 1,		CONFIG : 'N U T, 0, 0, 1',
	X =  178.000  mm,	Y =  61.000  mm,	Z =   0.600 mm,
	W =180.000 deg,	P =   0.000 deg,	R =    90.000 deg
};
P[3570]{
   GP1:
	UF : 1, UT : 1,		CONFIG : 'N U T, 0, 0, 1',
	X =  178.000  mm,	Y =  61.000  mm,	Z =   15.000 mm,
	W =180.000 deg,	P =   0.000 deg,	R =    90.000 deg
};
P[3571]{
   GP1:
	UF : 1, UT : 1,		CONFIG : 'N U T, 0, 0, 1',
	X =  1.000  mm,	Y =  64.000  mm,	Z =   15.000 mm,
	W =180.000 deg,	P =   0.000 deg,	R =    90.000 deg
};
P[3572]{
   GP1:
	UF : 1, UT : 1,		CONFIG : 'N U T, 0, 0, 1',
	X =  1.000  mm,	Y =  64.000  mm,	Z =   0.600 mm,
	W =180.000 deg,	P =   0.000 deg,	R =    90.000 deg
};
P[3573]{
   GP1:
	UF : 1, UT : 1,		CONFIG : 'N U T, 0, 0, 1',
	X =  1.000  mm,	Y =  64.000  mm,	Z =   15.000 mm,
	W =180.000 deg,	P =   0.000 deg,	R =    90.000 deg
};
P[3574]{
   GP1:
	UF : 1, UT : 1,		CONFIG : 'N U T, 0, 0, 1',
	X =  4.000  mm,	Y =  64.000  mm,	Z =   15.000 mm,
	W =180.000 deg,	P =   0.000 deg,	R =    90.000 deg
};
P[3575]{
   GP1:
	UF : 1, UT : 1,		CONFIG : 'N U T, 0, 0, 1',
	X =  4.000  mm,	Y =  64.000  mm,	Z =   0.600 mm,
	W =180.000 deg,	P =   0.000 deg,	R =    90.000 deg
};
P[3576]{
   GP1:
	UF : 1, UT : 1,		CONFIG : 'N U T, 0, 0, 1',
	X =  4.000  mm,	Y =  64.000  mm,	Z =   15.000 mm,
	W =180.000 deg,	P =   0.000 deg,	R =    90.000 deg
};
P[3577]{
   GP1:
	UF : 1, UT : 1,		CONFIG : 'N U T, 0, 0, 1',
	X =  7.000  mm,	Y =  64.000  mm,	Z =   15.000 mm,
	W =180.000 deg,	P =   0.000 deg,	R =    90.000 deg
};
P[3578]{
   GP1:
	UF : 1, UT : 1,		CONFIG : 'N U T, 0, 0, 1',
	X =  7.000  mm,	Y =  64.000  mm,	Z =   0.600 mm,
	W =180.000 deg,	P =   0.000 deg,	R =    90.000 deg
};
P[3579]{
   GP1:
	UF : 1, UT : 1,		CONFIG : 'N U T, 0, 0, 1',
	X =  7.000  mm,	Y =  64.000  mm,	Z =   15.000 mm,
	W =180.000 deg,	P =   0.000 deg,	R =    90.000 deg
};
P[3580]{
   GP1:
	UF : 1, UT : 1,		CONFIG : 'N U T, 0, 0, 1',
	X =  10.000  mm,	Y =  64.000  mm,	Z =   15.000 mm,
	W =180.000 deg,	P =   0.000 deg,	R =    90.000 deg
};
P[3581]{
   GP1:
	UF : 1, UT : 1,		CONFIG : 'N U T, 0, 0, 1',
	X =  10.000  mm,	Y =  64.000  mm,	Z =   0.600 mm,
	W =180.000 deg,	P =   0.000 deg,	R =    90.000 deg
};
P[3582]{
   GP1:
	UF : 1, UT : 1,		CONFIG : 'N U T, 0, 0, 1',
	X =  10.000  mm,	Y =  64.000  mm,	Z =   15.000 mm,
	W =180.000 deg,	P =   0.000 deg,	R =    90.000 deg
};
P[3583]{
   GP1:
	UF : 1, UT : 1,		CONFIG : 'N U T, 0, 0, 1',
	X =  13.000  mm,	Y =  64.000  mm,	Z =   15.000 mm,
	W =180.000 deg,	P =   0.000 deg,	R =    90.000 deg
};
P[3584]{
   GP1:
	UF : 1, UT : 1,		CONFIG : 'N U T, 0, 0, 1',
	X =  13.000  mm,	Y =  64.000  mm,	Z =   0.600 mm,
	W =180.000 deg,	P =   0.000 deg,	R =    90.000 deg
};
P[3585]{
   GP1:
	UF : 1, UT : 1,		CONFIG : 'N U T, 0, 0, 1',
	X =  13.000  mm,	Y =  64.000  mm,	Z =   15.000 mm,
	W =180.000 deg,	P =   0.000 deg,	R =    90.000 deg
};
P[3586]{
   GP1:
	UF : 1, UT : 1,		CONFIG : 'N U T, 0, 0, 1',
	X =  16.000  mm,	Y =  64.000  mm,	Z =   15.000 mm,
	W =180.000 deg,	P =   0.000 deg,	R =    90.000 deg
};
P[3587]{
   GP1:
	UF : 1, UT : 1,		CONFIG : 'N U T, 0, 0, 1',
	X =  16.000  mm,	Y =  64.000  mm,	Z =   0.600 mm,
	W =180.000 deg,	P =   0.000 deg,	R =    90.000 deg
};
P[3588]{
   GP1:
	UF : 1, UT : 1,		CONFIG : 'N U T, 0, 0, 1',
	X =  16.000  mm,	Y =  64.000  mm,	Z =   15.000 mm,
	W =180.000 deg,	P =   0.000 deg,	R =    90.000 deg
};
P[3589]{
   GP1:
	UF : 1, UT : 1,		CONFIG : 'N U T, 0, 0, 1',
	X =  19.000  mm,	Y =  64.000  mm,	Z =   15.000 mm,
	W =180.000 deg,	P =   0.000 deg,	R =    90.000 deg
};
P[3590]{
   GP1:
	UF : 1, UT : 1,		CONFIG : 'N U T, 0, 0, 1',
	X =  19.000  mm,	Y =  64.000  mm,	Z =   0.600 mm,
	W =180.000 deg,	P =   0.000 deg,	R =    90.000 deg
};
P[3591]{
   GP1:
	UF : 1, UT : 1,		CONFIG : 'N U T, 0, 0, 1',
	X =  19.000  mm,	Y =  64.000  mm,	Z =   15.000 mm,
	W =180.000 deg,	P =   0.000 deg,	R =    90.000 deg
};
P[3592]{
   GP1:
	UF : 1, UT : 1,		CONFIG : 'N U T, 0, 0, 1',
	X =  22.000  mm,	Y =  64.000  mm,	Z =   15.000 mm,
	W =180.000 deg,	P =   0.000 deg,	R =    90.000 deg
};
P[3593]{
   GP1:
	UF : 1, UT : 1,		CONFIG : 'N U T, 0, 0, 1',
	X =  22.000  mm,	Y =  64.000  mm,	Z =   0.600 mm,
	W =180.000 deg,	P =   0.000 deg,	R =    90.000 deg
};
P[3594]{
   GP1:
	UF : 1, UT : 1,		CONFIG : 'N U T, 0, 0, 1',
	X =  22.000  mm,	Y =  64.000  mm,	Z =   15.000 mm,
	W =180.000 deg,	P =   0.000 deg,	R =    90.000 deg
};
P[3595]{
   GP1:
	UF : 1, UT : 1,		CONFIG : 'N U T, 0, 0, 1',
	X =  25.000  mm,	Y =  64.000  mm,	Z =   15.000 mm,
	W =180.000 deg,	P =   0.000 deg,	R =    90.000 deg
};
P[3596]{
   GP1:
	UF : 1, UT : 1,		CONFIG : 'N U T, 0, 0, 1',
	X =  25.000  mm,	Y =  64.000  mm,	Z =   0.600 mm,
	W =180.000 deg,	P =   0.000 deg,	R =    90.000 deg
};
P[3597]{
   GP1:
